# B&R Automation Studio project mappFramework
Automation Studio 4.10.4.38 SP; technology packages: mapp 5.16.1, mappCockpit 5.16.0, mappControl 5.16.0, mappFramework 1.0.0, mappMotion 5.16.2, mappView 5.16.1

## Configuration PPC2200

### Task classes (Cpu.sw)
```
Cyclic#1 (cycle 1600 us, tolerance 1600 us):
  MainCtrl <- MainControl.MainCtrl.prg [disabled]
  AxisMgr <- MachineControl.AxisTemplate.AxisMgr.prg [disabled]
  AppAxis_1 <- MachineControl.AppAxis_1.AppAxis_1.prg
  CrossCutte <- MachineControl.CrossCutter.CrossCutter.prg [disabled]
Cyclic#2 (cycle 3200 us, tolerance 3200 us):
  PIDControl <- MainControl.PIDControl.prg [disabled]
Cyclic#5 (cycle 25600 us, tolerance 25600 us):
  ProcessCon <- Infrastructure.SysServices.ProcessConfig.prg [disabled]
  AlarmMgr <- Infrastructure.AlarmX.AlarmMgr.prg
  FileMgr <- Infrastructure.File.FileMgr.prg
  ReportMgr <- Infrastructure.Report.ReportMgr.prg
  AuditMgr <- Infrastructure.Audit.AuditMgr.prg
  UserXMgr <- Infrastructure.UserX.UserXMgr.prg
  DataMgr <- Infrastructure.Data.DataMgr.prg
  RecipeMgr <- Infrastructure.Recipe.RecipeMgr.prg
  UsbMgr <- Infrastructure.Usb.UsbMgr.prg
  BackupMgr <- Infrastructure.Backup.BackupMgr.prg
Cyclic#8 (cycle 9600 us):
  IoBrowser <- Infrastructure.SysServices.IoBrowser.prg
  SysServs <- Infrastructure.SysServices.SysServs.prg
DataObjects: McAcpSys
NcDataObjects: McDriveLog
Binaries: TCData, OpcUaSrv, McAcpSim, mCoWebSc, McProfGen, udbdef, TCLang, McAcpDrv, mvLoader, arsvcreg, arflatprv, FWRules, arcoal, sysconf, CutterAlm, asfw, UserXlogin, MachineGrp, Role, User, Settings, ashwd, ashwac, CutVirt, iomap, arconfig, CutAxis, CutCamAut, myUnits, CutterGrp, TC, BackupFile, Config, RecipeXML, AlarmXHist, RecipeCSV, VAppAxis1, Axis1Alm, Axis1Grp, AppAxis1, RecipeFile, DataFile, ReportFile, AuditFile, AuditCfg, FileCfg, BackupCfg, AlarmXCfg, ReportCfg, UserXCfg, DataCfg, Report, Audit, Data, Backup, UserX, AlarmX, Recipe, McMechSys, ConvVirt, ConvAxis, ConvGrp, ConvAlm, Cutter, AlmHistory, Rcp, Alarm, UsX
Libraries: operator, runtime, astime, AsIecCon, brsystem, sys_lib, AsArSdm, FileIO, standard, AsBrStr, asstring, AsBrWStr, ArUser, AsMem, AsARCfg, MTTypes, AsZip, DataObj, AsUPS, AsIO, AsIOMMan, Gat, IoMapMan, ArCfgMan, MTBasics, AsUSB, CoTrace, MpFile, MpData, MpBase, MpAxis, MpWebXs, MpAudit, MpRecipe, MpUserX, MpReport, MpAlarmX, MpCom, MpBackup, McAxis, McBase, McAcpAx, McPureVAx, McAcpPar, MpServer, MpRegMark, dvframe, AsIODiag, aseth, arssl, asepl, powerlnk, ashw, arproject, arcert, LoggingLib, snprintf, asarlog, asarprof
```

### Hardware
```
5AP1130.185C-000 : 5AP1130.185C-000 v2.0.0.0
5PPC2200_AL14_000 : 5PPC2200.AL14-000 v2.0.1.0  [SY -> 5AP1130.185C-000.SY1]
  Connector IF3:
    AssignedOperatingSystem = ARemb
    ActivateDevice = 1
    ActivateSnmp = 1
  Connector IF4:
    AssignedOperatingSystem = GPOS
  Connector IF7:
    OperatingSystem = ARemb
    ActivateDevice = 1
  Connector IF5:
    AssignedOperatingSystem = ARemb
  Connector IF6:
    AssignedOperatingSystem = GPOS
  ConfigurationID = mappFW_PPC2200
  UserPartitionSize = 128
  Simulation = 1
  SystemTick = 1600
  TaskClassIdleTime = 1600
  Cyclic1Duration = 1600
  Cyclic1Tolerance = 1600
  Cyclic2Duration = 3200
  Cyclic2Tolerance = 3200
  Cyclic3Duration = 6400
  Cyclic3Tolerance = 6400
  Cyclic4Duration = 12800
  Cyclic4Tolerance = 12800
  Cyclic5Duration = 25600
  Cyclic5Tolerance = 25600
  Cyclic6Duration = 51200
  Cyclic6Tolerance = 51200
  Cyclic7Duration = 102400
  Cyclic7Tolerance = 102400
  Cyclic8Duration = 9600
  FileDevice1
  FileDeviceName1 = UserPartition
  FileDevicePath1 = F:\
  FileDevice2
  FileDeviceName2 = mappRecipeFiles
  FileDevicePath2 = F:\Recipe
  FileDevice3
  FileDeviceName3 = mappAuditFiles
  FileDevicePath3 = F:\Audit
  FileDevice4
  FileDeviceName4 = mappReportFiles
  FileDevicePath4 = F:\Report
  FileDevice5
  FileDeviceName5 = mappDataFiles
  FileDevicePath5 = F:\Data
  FileDevice6
  FileDeviceName6 = mappBackupFiles
  FileDevicePath6 = F:\Backup
  FileDevice7
  FileDeviceName7 = mappAlarmXFiles
  FileDevicePath7 = F:\AlarmX
  FileDevice8
  FileDeviceName8 = mappUserXFiles
  FileDevicePath8 = F:\UserX
  TimeZone = 65
  ActivateDaylightSavingTime = 1
  FtpUser1
  FtpUsername1 = user
  FtpUserPassword1 = sHpIbnZIAriJzdWitYyNPul7Ws1MiS3ggYkn5Z1jgCk=
  FtpUserSalt1 = 13A/KPuX
  FTPAccessRight1 = 0
  FTPdevice1 = ALL
  ActivateOpcUa = 1
  OpcUaInformationModels_PV_Version = 1
  ActivateHypervisor = 1
```

### VAppAxis1.purevaxcfg - 5PPC2200_AL14_000/mappMotion/AppAxis_1/VAppAxis1.purevaxcfg
```
Element gMpLinkPureVAxCfgAppAxis_1 (Type=purevaxcfg)
  TypeID = PureVAxConfig
  PureVAxis:
    AxisReference = gMpLinkAppAxis_1
    Homing:
      Mode = Direct
        Position = 0.0
        ReferencePulse = NotUsed
      RestorePositionVariable
    JerkFilter = NotUsed
```

### CutVirt.purevaxcfg - 5PPC2200_AL14_000/mappMotion/CrossCutter/CutVirt.purevaxcfg
```
Element PureVAxCfg_CrossCutter (Type=purevaxcfg)
  TypeID = PureVAxConfig
  PureVAxis:
    AxisReference = gAxisCrossCutter
    Homing:
      Mode = Direct
        Position = 0.0
        ReferencePulse = NotUsed
      RestorePositionVariable
    JerkFilter = NotUsed
```

### Axis1Grp.mpcomgroup - 5PPC2200_AL14_000/mappServices/AppAxis_1/Axis1Grp.mpcomgroup
```
Element gMpLinkGroupAppAxis_1 (Type=mpcomgroup)
  Linking:
    Subnodes:
      0 = gMpLinkAppAxis_1
      1 = gMpLinkAlarmXCoreAppAxis_1
  Alarms = MpAlarmX
```

### BackupFile.mpfilemanagerui - 5PPC2200_AL14_000/mappServices/Backup/BackupFile.mpfilemanagerui
```
Element gMpLinkFileManagerUIBackup (Type=mpfilemanagerui)
  Alarms = MpAlarmX
    mapp.AlarmX.Core.Configuration:
      [0]:
        Message = {$File/Alarms/DeviceNotFound}
      [1]:
        Message = {$File/Alarms/AlreadyExisting}
      [2]:
        Message = {$File/Alarms/FileSystemError}
```

### CutterGrp.mpcomgroup - 5PPC2200_AL14_000/mappServices/CrossCutter/CutterGrp.mpcomgroup
```
Element gGroupCutter (Type=mpcomgroup)
  Linking:
    Subnodes:
      0 = gAxisCrossCutter
      1 = gAlarmXCore_Cutter
  Alarms = MpAlarmX
```

### FileCfg.mpfilemanagerui - 5PPC2200_AL14_000/mappServices/File/FileCfg.mpfilemanagerui
```
Element gMpLinkFileManagerUIFile (Type=mpfilemanagerui)
  Alarms = MpAlarmX
    mapp.AlarmX.Core.Configuration:
      [0]:
        Message = {$File/Alarms/DeviceNotFound}
      [1]:
        Message = {$File/Alarms/AlreadyExisting}
      [2]:
        Message = {$File/Alarms/FileSystemError}
```

### RecipeXML.mprecipexml - 5PPC2200_AL14_000/mappServices/Recipe/RecipeXML.mprecipexml
```
Element gMpLinkRecipeXml (Type=mprecipexml)
  mapp.Recipe.Xml:
    Auditing = MpAudit
  Alarms = MpAlarmX
    mapp.AlarmX.Core.Configuration:
      [0]:
        Message = {$Recipe/Alarms/SaveFailed}
      [1]:
        Message = {$Recipe/Alarms/SaveFailedPartial}
        Disable = TRUE
      [2]:
        Message = {$Recipe/Alarms/LoadFailed}
      [3]:
        Message = {$Recipe/Alarms/LoadFailedPartial}
        Disable = TRUE
```

### ReportCfg.mpreportcore - 5PPC2200_AL14_000/mappServices/Report/ReportCfg.mpreportcore
```
Element gMpLinkReport (Type=mpreportcore)
  MpReport:
    Settings:
      ResourceDeviceName = mappReport
      LanguageDependent:
        [0]:
          Language = en
          Font = 1
        [1]:
          Language = zh-CN
    PageLayouts:
      [0]:
        Name = Default
    Styles:
      Text:
        [0]:
          Name = Default
          Size = 12
        [1]:
          Name = Header
          Style = 1
          Size = 20
          Color = FF9900
        [2]:
          Name = Subheader
          Size = 16
          Color = FF9900
      Table:
        [0]:
          Name = Default
          Padding = 10
      Line:
        [0]:
          Name = Default
          Color = FF9900
      Chart:
        PieChart:
          [0]:
            Name = Default
            BorderWidth = 0
        LineChart:
          [0]:
            Name = Default
        BarChart:
          [0]:
            Name = Default
    Tables:
      [0]:
        Name = Information
        TableStyle = Default
        TextStyle = Default
        [0]:
          [0] = TextId
            Source = RecipeName
            Width = 50
          [1] = ValueId
            Value:
              ProcessVariable = ::RecipeMgr:MpRecipe_0.Info.LastLoadedRecipe
            Width = 50
        [1]:
          [0] = TextId
            Source = Index
            Width = 50
          [1] = TextId
            Source = Length [mm]
            Width = 50
          [2] = TextId
            Source = Number
            Width = 50
        [2]:
          [0] = TextId
            Source = 1
            Width = 50
          [1] = ValueId
            Value:
              ProcessVariable = ::MainCtrl:MainCtrl.Para.ProductLength[0]
            Width = 50
          [2] = ValueId
            Value:
              ProcessVariable = ::MainCtrl:MainCtrl.Para.ProductNumber[0]
            Width = 50
        [3]:
          [0] = TextId
            Source = 2
            Width = 50
          [1] = ValueId
            Value:
              ProcessVariable = ::MainCtrl:MainCtrl.Para.ProductLength[1]
            Width = 50
          [2] = ValueId
            Value:
              ProcessVariable = ::MainCtrl:MainCtrl.Para.ProductNumber[1]
            Width = 50
        [4]:
          [0] = TextId
            Source = 3
            Width = 50
          [1] = ValueId
            Value:
              ProcessVariable = ::MainCtrl:MainCtrl.Para.ProductLength[2]
            Width = 50
          [2] = ValueId
            Value:
              ProcessVariable = ::MainCtrl:MainCtrl.Para.ProductNumber[2]
            Width = 50
        [5]:
          [0] = TextId
            Source = 4
            Width = 50
          [1] = ValueId
            Value:
              ProcessVariable = ::MainCtrl:MainCtrl.Para.ProductLength[3]
            Width = 50
          [2] = ValueId
            Value:
              ProcessVariable = ::MainCtrl:MainCtrl.Para.ProductNumber[3]
            Width = 50
        [6]:
          [0] = TextId
            Source = 5
            Width = 50
          [1] = ValueId
            Value:
              ProcessVariable = ::MainCtrl:MainCtrl.Para.ProductLength[4]
            Width = 50
          [2] = ValueId
            Value:
              ProcessVariable = ::MainCtrl:MainCtrl.Para.ProductNumber[4]
            Width = 50
    Contents:
      [0]:
        Name = ContentHeader
        [0]:
          Text = {Header}
        [1] = DateTime
        [2] = Line
          LineStyle = Default
      [1]:
        Name = ContentTable
        [0] = Table
          Table = Information
          HorizontalAlign = 1
      [2]:
        Name = Header
        [0]:
          Text = Report of the Cross Cutter Machine
          HorizontalAlign = 1
          TextStyle = Header
      [3]:
        Name = EmptyLine
        [0] = EmptyLine
      [4]:
        Name = Underline
        [0] = Line
          LineStyle = Default
      [5]:
        Name = Date
        [0] = DateTime
          TextStyle = Default
    Reports:
      [0]:
        Name = Report
        PageLayout = Default
        Header = Header
        [0]:
          [0]:
            Content = Underline
        [1]:
          [0]:
            Content = EmptyLine
        [2]:
          Heading:
            Text = Time
            TextStyle = Subheader
          [0]:
            Content = Date
        [3]:
          [0]:
            Content = EmptyLine
        [4]:
          [0]:
            Content = EmptyLine
        [5]:
          Heading:
            Text = Data
            TextStyle = Subheader
          [0]:
            Content = ContentTable
  Alarms = MpAlarmX
    mapp.AlarmX.Core.Configuration:
      [0]:
        Message = {$Report/Alarms/GenerateFailed}
```

## Configuration TS_UnitTest_Sample

CPU , AutomationRuntime D4.91, Build 6.3.0, Safety 0.0

### Hardware
```
PC_any : PC_any v1.1.1.0 (OrderNumber=PC)
  ConfigurationID = GAT_TS_UnitTest_Sample
  Cyclic1Duration = 10000
  Cyclic8Duration = 10000
  ActivateOpcUa = 1
  OpcUaInformationModels_PV_Version = 1
```

### AxisTest.vvm - PC_any/AxisTest.vvm
```iecst
VAR_CONFIG
	::prototypeT:AxisControl.Command AT %Q.::AxisContro:AxisControl.Command; (*Insert your comment here...*)
	::prototypeT:AxisControl.Parameters AT %Q.::AxisContro:AxisControl.Parameters; (*Insert your comment here...*)
	::AxisContro:AxisControl.Status AT %Q.::prototypeT:AxisControl.Status; (*Insert your comment here...*)
END_VAR
```

### Cutter.regmarkdetection - PC_any/mappControl/Cutter.regmarkdetection
```
Element gRegMarkDetection_Cutter (Type=regmarkdetection)
  RegistrationMarkDetection:
    SensorSignal:
      AxisReference = gAxisCrossCutter
      DelayCompensation:
        AdditionalDelayTime  // 0.
    Measurement = MarkToCylinder
      Product:
        Position:
          AxisReference = gAxisAppAxis_1
          Source = SetValue
        Length:
          Value = 70
    Detection = MiddleOfEdges
      SetMarkPosition = 0
      ExpectationWindow:
        Width = 25
      MarkWidthMonitoring:
        MinimumWidth = 7
        MaximumWidth = 15
      MissedMarkReaction:
        MarkPosition = LastValue
        AutomaticSearch = Used
          AdditionalExpectationWindowShift = 25
    OutputSignals:
      ActualMarkPosition = ::CrossCutte:RegistrationControl.ActualMarkPosition
      MarkPositionError = ::CrossCutte:RegistrationControl.MarkPositionError
      ActualProductLength = ::CrossCutte:RegistrationControl.ActualProductLength
      ActualIntervalLength = ::CrossCutte:RegistrationControl.ActualIntervalLength
  Alarms = MpAlarmX
```

### TestAlm.mpalarmxcore - PC_any/mappServices/AxisTest/TestAlm.mpalarmxcore
```
Element gAlarmXCore_Test (Type=mpalarmxcore)
  mapp.AlarmX.Core:
    BySeverity:
      [0]:
        Severity = 1..9
        [0] = Reaction
          Name = Info
        [1] = Escalate
      [1]:
        Severity = 10..19
        [0] = Reaction
          Name = Error
        [1] = Escalate
      [2]:
        Severity = 20..29
        [0] = Reaction
          Name = Error
        [1] = Escalate
        [2] = EscalateReaction
          Reaction = Error
      [3]:
        Severity = 30..39
        [0] = Reaction
          Name = Safety
        [1] = Escalate
        [2] = Remain
    Default:
      [0] = Reaction
        Name = Duplicate
      [1] = Escalate
      [2] = Remain
  mapp.AlarmX.Core.Configuration:
    [0]:
      Name = ReferenceRequired
      Message = {$IAT/Axis/Info/Name} : {$IAT/Axis/Alarms/ReferenceRequired}
      Severity = 10
      Behavior = DiscreteValueMonitoring
        Monitoring:
          MonitoredPV = ::AxisContro:AxisControl.Status.ReferenceRequired
          TriggerValues:
            [0] = 1
```

## Logical view

Binary libraries used (declarations not repeated): UtMgr 2.01.0, UtWs 2.01.0, ArCfgMan 1.01.1, ArUser, AsARCfg, AsBrStr, AsBrWStr, AsIecCon, AsIO, AsIODiag, AsIOMMan, asstring, AsUPS, AsUSB, AsZip, brsystem, CoTrace, DataObj, dvframe, FileIO, IoMapMan 1.01.1, McAcpAx 5.16.2, McAcpPar 5.16.2, McAxis, McPureVAx 5.16.2, MpAlarmX 5.16.1, MpAudit 5.16.1, MpAxis, MpBackup 5.16.1, MpBase 5.16.0, MpCom 5.16.1, MpData 5.16.1, MpFile 5.16.1, MpRecipe, MpRegMark 5.16.0, MpReport 5.16.1, MpServer 5.16.0, MpUserX 5.16.1, MpWebXs 5.16.1, MTBasics 5.16.0, MTTypes 1.03.4, operator, runtime, standard, sys_lib

### mappFrameworkGlobal.var
```iecst
VAR CONSTANT
	PARAMETERS_CATEGORY : STRING[10] := 'Parameters'; (*Recipe category for runtime parameters*)
	MACHINE_CONFIGURATION_CATEGORY : STRING[30] := 'Machine Configuration'; (*Recipe category for machine configuration settings*)
	MAX_IDX_USB_DEV_LIST : USINT := 1; (*Maximum number of USB storage devices. Value 1 = 2 USB devices (index 0 and 1)*)
END_VAR
VAR
	gUSBAvailable : ARRAY[0..MAX_IDX_USB_DEV_LIST] OF BOOL; (*Boolean array for whether the USB device is plugged in*)
END_VAR
```

- Project.language (not shown)

### Program Logical/Infrastructure/AlarmX/AlarmMgr (IEC) - Alarm manager

#### ExecuteQuery.st
```iecst
ACTION ExecuteQuery:

	// Initialize mapp function block
	QueryActiveAlarms_0.MpLink := ADR(gMpLinkAlarmXCore);
	QueryActiveAlarms_0.Enable := TRUE;
	QueryActiveAlarms_0.Name := ADR('ActiveAlarms');
	QueryActiveAlarms_0.Language := ADR('en');
	QueryActiveAlarms_0();

	CASE (AlarmQuery.State) OF
		ACTIVE_ALARM_WAIT:
			// Wait until the RunQuery command is triggered from the HMI.
			// If you prefer that the query runs anytime new data is available, then uncomment line 15 and comment out line 16 and delete
			// the "Run query" button from the HMI.
			//IF (AlarmQuery.LastUpdateCount <> AlarmQuery.UpdateCount) THEN
			IF (HmiAlarmX.Commands.RunQuery = TRUE) THEN
				brsmemset(ADR(AlarmQuery.Alarms[0]), 0, SIZEOF(AlarmQuery.Alarms));
				AlarmQuery.LastUpdateCount := AlarmQuery.UpdateCount;
				QueryActiveAlarms_0.Execute := TRUE;
				HmiAlarmX.Commands.RunQuery := FALSE;
				AlarmQuery.State := ACTIVE_ALARM_QUERY;
			END_IF

		ACTIVE_ALARM_QUERY:
			// If the number of query results is less than MAX_QUERY_RESULTS, return to the wait state
			IF ((QueryActiveAlarms_0.CommandDone = TRUE) AND (QueryActiveAlarms_0.Info.HasMoreRows = FALSE)) THEN
				QueryActiveAlarms_0.Execute := FALSE;
				QueryActiveAlarms_0.Next := FALSE;
				AlarmQuery.State := ACTIVE_ALARM_WAIT;
				// If the number of query results is more than MAX_QUERY_RESULTS, then query the next set of results
			ELSIF ((QueryActiveAlarms_0.CommandDone = TRUE) AND (QueryActiveAlarms_0.Info.HasMoreRows = TRUE)) THEN
				QueryActiveAlarms_0.Next := FALSE;
				AlarmQuery.State := ACTIVE_ALARM_NEXT;
			END_IF

		ACTIVE_ALARM_NEXT:
			IF (AlarmQuery.Next = TRUE) THEN
				// By default, AlarmQuery.Alarms has 20 elements, so it can hold 20 query results at a time (MAX_QUERY_RESULTS = 19).
				// If AlarmQuery.Next is true, this means the query result is more than 20 alarms.
				// If you want to save the data for the first 20 alarms, add code here to copy AlarmQuery.Alarms to another location.
				// Otherwise, the older alarms in the query will get overwritten with the newest entries here.
				brsmemset(ADR(AlarmQuery.Alarms[0]), 0, SIZEOF(AlarmQuery.Alarms));
				AlarmQuery.Next := FALSE;
				QueryActiveAlarms_0.Next := TRUE;
				AlarmQuery.State := ACTIVE_ALARM_QUERY;
			END_IF
	END_CASE

	// Convert the query results into arrays that can easily be bound to the Table widget in mapp View
	FOR i := 0 TO MAX_QUERY_RESULTS DO
		HmiAlarmX.Status.Query.Active[i] := AlarmQuery.Alarms[i].Active;
		HmiAlarmX.Status.Query.Acknowledged[i] := AlarmQuery.Alarms[i].Acknowledged;
		HmiAlarmX.Status.Query.Scope[i] := AlarmQuery.Alarms[i].Scope;
		HmiAlarmX.Status.Query.Name[i] := AlarmQuery.Alarms[i].Name;
		HmiAlarmX.Status.Query.Message[i] := AlarmQuery.Alarms[i].Message;
		HmiAlarmX.Status.Query.AdditionalInfo[i] := AlarmQuery.Alarms[i].AdditionalInfo;
		HmiAlarmX.Status.Query.TimeStamp[i] := AlarmQuery.Alarms[i].TimeStamp;
		HmiAlarmX.Status.Query.Severity[i] := AlarmQuery.Alarms[i].Severity;
	END_FOR

END_ACTION
```

- Program Logical/Infrastructure/Audit/AuditMgr (IEC) (no source held here)

### Program Logical/Infrastructure/Backup/BackupMgr (IEC) - Backup manager

#### BackupMgr.typ
```iecst
(*Structure types*)

TYPE
	BackupHmiInterfaceType : 	STRUCT  (*HMI interface structure*)
		Commands : BackupHmiCommandsType; (*Structure to hold the commands from the HMI*)
		Parameters : BackupHmiParametersType; (*Structure to hold the parameters for the HMI*)
		Status : BackupHmiStatusType; (*Structure to hold the status information from the HMI*)
	END_STRUCT;
	BackupHmiCommandsType : 	STRUCT  (*Structure to hold the commands from the HMI*)
		Create : BOOL; (*Create a backup*)
		Restore : BOOL; (*Restore a backup*)
		Delete : BOOL; (*Delete a backup*)
		SaveConfig : BOOL; (*Save automatic backup configuration settings*)
		Reset : BOOL; (*Error reset*)
	END_STRUCT;
	BackupHmiParametersType : 	STRUCT  (*Structure to hold the parameters for the HMI*)
		Name : STRING[80] := 'myBackup'; (*Name of the backup*)
		AutomaticBackup : AutomaticBackupType; (*Automatic backup settings*)
	END_STRUCT;
	BackupHmiStatusType : 	STRUCT  (*Structure to hold the status information from the HMI*)
		Busy : BOOL; (*Backup is busy executing an action*)
		Error : BOOL; (*Error flag*)
		CreateAllowed : BOOL; (*Bit to indicate it is allowable to create a backup right now*)
		RestoreAllowed : BOOL; (*Bit to indicate it is allowable to restore a backup right now*)
		FileNames : ARRAY[0..49]OF STRING[80]; (*Existing backup file names*)
		TimeStamps : ARRAY[0..49]OF DATE_AND_TIME; (*Time stamps for existing backups*)
		Size : {REDUND_UNREPLICABLE} ARRAY[0..49]OF UDINT; (*Sizes of existing backup files*)
		Info : MpBackupProjectInfoRequestType; (*Project information (name, configuration ID, configuration version)*)
		DeviceDataProvider : ARRAY[0..MAX_IDX_FILE_DEV]OF STRING[100]; (*Data provider for file device dropdown on automatic backup configuration pop-up*)
		TableConfig : ARRAY[0..1]OF STRING[120]; (*Table configuration for the list of available backups*)
		SimulationActive : BOOL; (*Flag for if simulation is active*)
		SelectedIndex : USINT; (*Index of the selected backup file*)
		LastSelectedIndex : USINT; (*Index of the last selected backup file*)
		LastSelectedDeviceIndex : UINT; (*Index of the last selected file device. Compared with MpFileManagerUIConnect.DeviceList.SelectedIndex*)
	END_STRUCT;
	AutomaticBackupType : 	STRUCT  (*Automatic backup settings*)
		Enable : BOOL; (*Enable automatic backup feature*)
		Prefix : STRING[50]; (*Name prefix for each automatic backup file*)
		Device : STRING[255]; (*File device to store the automatic backup*)
		Mode : AutomaticBackupModeType; (*Automatic backup time interval*)
		OverwriteOldest : MpBackupOverwriteOldestType; (*Defines whether older backups should be deleted or not*)
	END_STRUCT;
	AutomaticBackupModeType : 	STRUCT  (*Automatic backup time interval*)
		Interval : AutomaticBackupIntervalEnum; (*Day interval (daily, or a specfiic day of the week)*)
		Hour : USINT; (*Time (hour)*)
		Minute : USINT; (*Time (minutes)*)
	END_STRUCT;
END_TYPE

(*Enumerations*)

TYPE
	AutomaticBackupIntervalEnum :
		( (*Selection for how often to automatically create a backup*)
		BACKUP_EVERYDAY, (*Every day*)
		BACKUP_MONDAY, (*Every Monday*)
		BACKUP_TUESDAY, (*Every Tuesday*)
		BACKUP_WEDNESDAY, (*Every Wednesday*)
		BACKUP_THURSDAY, (*Every Thursday*)
		BACKUP_FRIDAY, (*Every Friday*)
		BACKUP_SATURDAY, (*Every Saturday*)
		BACKUP_SUNDAY (*Every Sunday*)
		);
	BackupStateEnum :
		( (*States for backup state machine*)
		BACKUP_IDLE, (*Wait state*)
		BACKUP_CREATING, (*Creating a backup*)
		BACKUP_RESTORING, (*Restoring a backup*)
		BACKUP_DELETING, (*Deleting a backup*)
		BACKUP_ERROR (*Error state*)
		);
END_TYPE
```

#### ChangeConfiguration.st
```iecst
ACTION ChangeConfiguration:

    MpBackupCoreConfig_0.MpLink := ADR(gMpLinkBackupCore);
    MpBackupCoreConfig_0.Configuration := ADR(MpBackupConfiguration);
    IF (MpBackupCoreConfig_0.Error = TRUE) THEN
        // Loading currently always throws an error about failed to write Auditing.Type
        IF (MpBackupCoreConfig_0.StatusID = mpBACKUP_ERR_CONFIG_LOAD) THEN
            LoadBackupConfiguration;
        END_IF

        MpBackupCoreConfig_0.Load := FALSE;
        MpBackupCoreConfig_0.Save := FALSE;
        MpBackupCoreConfig_0.ErrorReset := TRUE;
    END_IF
    MpBackupCoreConfig_0();
    MpBackupCoreConfig_0.ErrorReset := FALSE;
    IF (MpBackupCoreConfig_0.CommandDone = TRUE) THEN
        IF (MpBackupCoreConfig_0.Load = TRUE) THEN
            LoadBackupConfiguration;
        END_IF
        MpBackupCoreConfig_0.Load := FALSE;
        MpBackupCoreConfig_0.Save := FALSE;
    END_IF

END_ACTION
```

### Program Logical/Infrastructure/Data/DataMgr

#### DataMgr.st
```iecst
//*********************************************************************************
//* Copyright: B&R Industrial Automation GmbH
//* Author:    B&R Industrial Automation GmbH
//* Created:   30. Sep 2020/08:00
//* Description: Tasks FOR Data Management control. The Data Management handling is done in this task.
//*********************************************************************************

PROGRAM _INIT

	// Create folder for this component on the user file device
	DirCreate_0(enable := TRUE, pDevice := ADR('UserPartition'), pName := ADR(LOCAL_FOLDER));

	// Check if folder already exist and if so disabled the function block call
	IF DirCreate_0.status = fiERR_DIR_ALREADY_EXIST THEN
		DirCreate_0(enable := FALSE);
	END_IF

	// Init mapp function blocks
	MpFileManagerUI_0.Enable := TRUE;
	MpFileManagerUI_0.MpLink := ADR(gMpLinkFileManagerUIData);
	MpFileManagerUI_0.UIConnect := ADR(MpFileManagerUIConnect);

	MpDataRecorder_0.MpLink := ADR(gMpLinkDataRecorder);
	MpDataRecorder_0.Enable := TRUE ;
	MpDataRecorder_0.DeviceName := ADR('mappDataFiles');
	MpDataRecorder_0.RecordMode := mpDATA_RECORD_MODE_TIME;
	MpDataRecorder_0.SamplingTime := t#5s;

	// Register PVs for data recording
	MpDataRegPar_x[0].MpLink := ADR(gMpLinkDataRecorder);
	MpDataRegPar_x[0].Enable := TRUE;
	MpDataRegPar_x[0].PVName := ADR('PIDControl:rActValue');
	MpDataRegPar_x[0].Description := ADR('Control Value');

	MpDataRegPar_x[1].MpLink := ADR(gMpLinkDataRecorder);
	MpDataRegPar_x[1].Enable := TRUE;
	MpDataRegPar_x[1].PVName := ADR('MainCtrl:MpAxisBasic_x[0].Velocity');
	MpDataRegPar_x[1].Description := ADR('Feeder Velocity');

	// Filter files for pdf type
	MpFileManagerUIConnect.File.Filter := '*.pdf';
END_PROGRAM

PROGRAM _CYCLIC
	//***************************************************
	FOR i := 0 TO 49 DO
		// Save Filenames to a seperate array for display in Table
		DisplayFileName[i] := MpFileManagerUIConnect.File.List.Items[i].Name;
		// Mark file selection
		MpFileManagerUIConnect.File.List.Items[i].IsSelected := (DisplayFileNameIndex = INT_TO_USINT(i));
    END_FOR
    // String for pdfViewer to display right report
	StrSelectedFile := CONCAT(STR_FILE_DEVICE, MpFileManagerUIConnect.File.List.Items[DisplayFileNameIndex].Name);

	// Configure visible file list
	brsstrcpy(ADR(TableConfig), ADR('{ "specRows": [{"from":'));
	brsitoa(MpFileManagerUIConnect.File.PathInfo.FileCount, ADR(TableConfig) + brsstrlen(ADR(TableConfig)));
	brsstrcat(ADR(TableConfig),  ADR(',"to":49, "visible":false}]}'));

	// Call function blocks
	MpDataRecorder_0();
	FOR i := 0 TO MAX_IDX_DATA_REG DO
		MpDataRegPar_x[i]();
	END_FOR
	MpFileManagerUI_0();

	// Reset ErrorReset command
	IF NOT MpDataRecorder_0.Error THEN
		MpDataRecorder_0.ErrorReset := FALSE;
	END_IF
	FOR i := 0 TO MAX_IDX_DATA_REG DO
		IF NOT MpDataRegPar_x[i].Error THEN
			MpDataRegPar_x[i].ErrorReset := FALSE;
		END_IF
	END_FOR
END_PROGRAM

PROGRAM _EXIT
	// Call mapp function blocks with enable = false
	MpFileManagerUI_0.Enable := FALSE;
	MpFileManagerUI_0();
	MpDataRecorder_0.Enable := FALSE;
	MpDataRecorder_0();
	FOR i := 0 TO MAX_IDX_DATA_REG DO
		MpDataRegPar_x[i].Enable := FALSE;
		MpDataRegPar_x[i]();
	END_FOR
END_PROGRAM
```

### Program Logical/Infrastructure/File/FileMgr (IEC)

#### FileMgr.typ - Local data types
```iecst
(*Structure types*)

TYPE
	FileHmiInterfaceType : 	STRUCT  (*Structure to hold commands, parameters and status from the HMI*)
		Commands : FileHmiCommandsType; (*Structure to hold the commands from the HMI*)
		Parameters : FileHmiParametersType; (*Structure to hold parameters for the mapp View HMI*)
		Status : FileHmiStatusType; (*Structure to hold status information from the mapp View HMI*)
	END_STRUCT;
	FileHmiCommandsType : 	STRUCT  (*Structure to hold the commands from the HMI*)
		Delete : BOOL; (*Delete file*)
		FolderUp : BOOL; (*Move back/up a folder*)
		EnterFolder : BOOL; (*Move forward/down a folder*)
		MultiSelect : BOOL; (*Enables the ability to select multiple files*)
		CheckFolder : BOOL; (*Run the FIFO check to determine if old files should be deleted*)
	END_STRUCT;
	FileHmiParametersType : 	STRUCT  (*Structure to hold parameters for the mapp View HMI*)
		OldSortOrder : MpFileManagerUISortOrderEnum; (*Previous sord order*)
		Fifo : FileHmiParaFifoType; (*Parameters for the FIFO feature (first-in-first-out)*)
	END_STRUCT;
	FileHmiStatusType : 	STRUCT  (*Structure to hold status information from the mapp View HMI*)
		FileNames : ARRAY[0..49]OF STRING[80]; (*List of file names*)
		TimeStamps : ARRAY[0..49]OF DATE_AND_TIME; (*List of time stamps for file names*)
		Type : ARRAY[0..49]OF DINT; (*List of file types*)
		Size : ARRAY[0..49]OF UDINT; (*List of file sizes*)
		DeviceDataProvider : ARRAY[0..MAX_IDX_FILE_DEV]OF STRING[100]; (*Data provider for the file device selector*)
		DeviceName : STRING[50]; (*File device name*)
		FileName : STRING[255]; (*Fille name*)
		TableConfig : ARRAY[0..1]OF STRING[120]; (*Table configuration for the file explorer (table widget) on the mapp View HMI*)
		IsFolder : BOOL; (*Flag for whether the item is a folder (versus a file)*)
		BackButton : BOOL; (*Flag for whether the back button should be shown*)
		DeleteStep : FileDeleteStepEnum; (*Enumeration for automatic file deletion steps*)
		AutoDeleteSelected : USINT; (*Number of selected items*)
		FolderSize : REAL; (*Size of currently selected folder*)
		SelectedIndex : USINT; (*Selected index in the file list*)
		CurrentPage : STRING[80]; (*Current page*)
	END_STRUCT;
	FileHmiParaFifoType : 	STRUCT  (*Parameters for the FIFO feature (first-in-first-out)*)
		Enable : BOOL; (*FIFO enable*)
		DeviceName : STRING[50]; (*File device that the FIFO is active on*)
		FifoType : FileFifoTypeEnum; (*Defines the delete behavior of the FIFO*)
		ScanInterval : DINT := 60; (*[minutes]*)
		MaxFileAge : UINT := 365; (*[days] Files older than 1 year will be deleted*)
		MaxFolderSize : REAL := 1000; (*[kB] - Max size of files inside the active folder*)
		MaxNumberOfFiles : UINT := 20; (*Max number of files inside active folder*)
	END_STRUCT;
	FilePathCheckType : 	STRUCT  (*Setup for checking available folders / file devices for FIleManager*)
		Folder : ARRAY[0..9]OF STRING[20]; (*Folder name in user partition*)
		DeviceList : MpFileManagerUIDeviceListType; (*Device name*)
	END_STRUCT;
END_TYPE

(*Enumerations*)

TYPE
	FileDeleteStepEnum :
		( (*Enumeration for file deletion steps*)
		FILE_DELETE_WAIT := 0, (*Wait state*)
		FILE_SCAN_FOLDER_WAIT, (*Wait for check for old files command*)
		FILE_SELECT_DEVICE, (*Switch file device to the configured one *)
		FILE_SORT_BY_DATE, (*Sort by date so the oldest files are at the end*)
		FILE_SORT_BY_DATE_WAIT, (*Wait step switching sorting mode*)
		FILE_CHECK_FOR_FILTER, (*Check which delete filter is active*)
		FILE_SELECT_OLDEST_FILES_0, (*Scan and select all file over the filter setting*)
		FILE_CALC_FOLDER_SIZE, (*Calculate the overall file size in the open folder*)
		FILE_SELECT_OLDEST_FILES_1, (*Scan and select all file over the filter setting*)
		FILE_DELETE_FILES, (*Set command to delete the selected oldest files*)
		FILE_CONFIRM_DELETE, (*Confirm the file delete*)
		FILE_RESET_SORT_BY, (*Restore old sort order*)
		FILE_RESET_SORT_BY_WAIT (*Waiting for restore previous sort order*)
		);
	FileFifoTypeEnum :
		( (*Defines the delete behavior of the FIFO*)
		FILE_FIFO_NUM_OF_FILES := 0, (*Delete according to total number of files*)
		FILE_FIFO_SIZE_OF_FOLDER (*Delete according to maximum folder size*)
		);
	FileTypeEnum :
		( (*Defines the type of file in order to update the displayed icon*)
		FOLDER := 0, (*Folder*)
		FILE := 1, (*File*)
		FILE_SELECTED := 2 (*The selected file*)
		);
END_TYPE
```

#### HMIActions.st - Supporting code for the HMI interface
```iecst
ACTION FormatDeviceDataProvider:

	// Select CF device if USB device is not available
    FOR i := 0 TO MAX_IDX_USB_DEV_LIST DO
        IF gUSBAvailable[i] THEN

			HmiFile.Status.DeviceDataProvider[i + USBOffset] := '{"value":"USB';
            brsitoa(i + 1, ADR(HmiFile.Status.DeviceDataProvider[i + USBOffset]) + brsstrlen(ADR(HmiFile.Status.DeviceDataProvider[i + USBOffset])));

			brsstrcat(ADR(HmiFile.Status.DeviceDataProvider[i + USBOffset]), ADR('","text":"USB'));
            brsitoa(i + 1, ADR(HmiFile.Status.DeviceDataProvider[i + USBOffset]) + brsstrlen(ADR(HmiFile.Status.DeviceDataProvider[i + USBOffset])));
            brsstrcat(ADR(HmiFile.Status.DeviceDataProvider[i + USBOffset]), ADR('"}'));

			PathCheck.DeviceList.DeviceNames[i + USBOffset] := 'USB';
			brsitoa(i + 1, ADR(PathCheck.DeviceList.DeviceNames[i + USBOffset]) + brsstrlen(ADR(PathCheck.DeviceList.DeviceNames[i + USBOffset])));
        ELSE
			brsmemset(ADR(HmiFile.Status.DeviceDataProvider[i + USBOffset]), 0, SIZEOF(HmiFile.Status.DeviceDataProvider[i + USBOffset]));
            brsmemset(ADR(PathCheck.DeviceList.DeviceNames[i + USBOffset]), 0, SIZEOF(PathCheck.DeviceList.DeviceNames[i + USBOffset]));
        END_IF
    END_FOR

	//Check initilized folder for existance and remove any from the device list that don't exist
	IF DirInfo_0.status = ERR_OK  THEN
		IF PathCheck.DeviceList.DeviceNames[DeviceListCount] = '' THEN
			//Delete entries past the actual number of devices found
			FOR i:=Index TO 9 DO
				MpFileManagerUIConnect.DeviceList.DeviceNames[i] := '';
			END_FOR
			Index := -1;
			DeviceListCount := -1;
		END_IF
		// copy device name from source list into the actual device list
		MpFileManagerUIConnect.DeviceList.DeviceNames[Index] := PathCheck.DeviceList.DeviceNames[DeviceListCount];
		Index := Index + 1;

		DeviceListCount := DeviceListCount + 1;
		IF DeviceListCount > 9 THEN
			DeviceListCount := 0;
		END_IF
		IF Index > 9 THEN
			Index := 0;
		END_IF
	ELSIF DirInfo_0.status = fiERR_DIR_NOT_EXIST  THEN
		DeviceListCount := DeviceListCount + 1;
		IF DeviceListCount > 9 THEN
			DeviceListCount := 0;
		END_IF
	END_IF

	DirInfo_0(enable:= TRUE, pDevice := ADR('UserPartition'), pPath := ADR(PathCheck.Folder[DeviceListCount]));

	// Configure visible device list
	HmiFile.Status.TableConfig[0] := '{ "specRows": [{"from":';
	FOR i := 0 TO 9 DO
		IF MpFileManagerUIConnect.DeviceList.DeviceNames[i] <> '' THEN
			DeviceCount := i + 1;
		END_IF
	END_FOR
	brsitoa((DeviceCount), ADR(HmiFile.Status.TableConfig[0]) + brsstrlen(ADR(HmiFile.Status.TableConfig[0])));
    brsstrcat(ADR(HmiFile.Status.TableConfig[0]),  ADR(',"to":9, "visible":false}]}'));

    // Configure visible file list
	HmiFile.Status.TableConfig[1] := '{ "specRows": [{"from":';
    brsitoa((MpFileManagerUIConnect.File.PathInfo.FileCount + MpFileManagerUIConnect.File.PathInfo.FolderCount), ADR(HmiFile.Status.TableConfig[1]) + brsstrlen(ADR(HmiFile.Status.TableConfig[1])));
    brsstrcat(ADR(HmiFile.Status.TableConfig[1]),  ADR(',"to":49, "visible":false}]}'));

END_ACTION

ACTION FileManager:

    MpFileManagerUI_0.MpLink := ADR(gMpLinkFileManagerUIFile);
    MpFileManagerUI_0.UIConnect := ADR(MpFileManagerUIConnect);
	MpFileManagerUI_0();

    FOR i := 0 TO ((SIZEOF(HmiFile.Status.FileNames)/SIZEOF(HmiFile.Status.FileNames[0])) - 1) DO
        HmiFile.Status.FileNames[i] := MpFileManagerUIConnect.File.List.Items[i].Name;
        HmiFile.Status.TimeStamps[i] := MpFileManagerUIConnect.File.List.Items[i].LastModified;
        HmiFile.Status.Size[i] := REAL_TO_UDINT(UDINT_TO_REAL(MpFileManagerUIConnect.File.List.Items[i].Size) * 0.001);

		// Set image array based on item type
		IF MpFileManagerUIConnect.File.List.Items[i].IsFolder THEN
			HmiFile.Status.Type[i] := FOLDER;
		ELSIF NOT MpFileManagerUIConnect.File.List.Items[i].IsFolder AND MpFileManagerUIConnect.File.List.Items[i].IsSelected THEN
			HmiFile.Status.Type[i] := FILE_SELECTED;
		ELSE
			HmiFile.Status.Type[i] := FILE;
		END_IF

		// Set file selected when the table is clicked Single and MultiSelect
		IF HmiFile.Status.DeleteStep = FILE_DELETE_WAIT THEN
			IF (MpFileManagerUIConnect.File.MultiSelect = FALSE) THEN
				IF (i = HmiFile.Status.SelectedIndex) THEN
					MpFileManagerUIConnect.File.List.Items[i].IsSelected := TRUE;
				ELSE
					MpFileManagerUIConnect.File.List.Items[i].IsSelected := FALSE;
				END_IF
			ELSIF (MpFileManagerUIConnect.File.MultiSelect = TRUE) AND HmiFile.Commands.MultiSelect THEN
				IF (i = HmiFile.Status.SelectedIndex) AND NOT MpFileManagerUIConnect.File.List.Items[i].IsSelected THEN
					MpFileManagerUIConnect.File.List.Items[i].IsSelected := TRUE;
					HmiFile.Commands.MultiSelect := FALSE;
				ELSIF (i = HmiFile.Status.SelectedIndex) AND MpFileManagerUIConnect.File.List.Items[i].IsSelected THEN
					MpFileManagerUIConnect.File.List.Items[i].IsSelected := FALSE;
					HmiFile.Commands.MultiSelect := FALSE;
				END_IF
			END_IF
		END_IF
    END_FOR

	// Read currently selected device name for HMI
	HmiFile.Status.DeviceName := MpFileManagerUIConnect.DeviceList.DeviceNames[MpFileManagerUIConnect.DeviceList.SelectedIndex];

	// Read if current selected object is folder
	HmiFile.Status.IsFolder := MpFileManagerUIConnect.File.List.Items[HmiFile.Status.SelectedIndex].IsFolder;

	// Control the folder structure when entering and leaving folders
	IF (HmiFile.Commands.EnterFolder) AND MpFileManagerUIConnect.File.List.Items[HmiFile.Status.SelectedIndex].IsFolder THEN
		HmiFile.Commands.EnterFolder := FALSE;
		MpFileManagerUIConnect.File.EnterFolder := TRUE;
		FolderDepthCount := FolderDepthCount + 1;
	ELSE
		HmiFile.Commands.EnterFolder := FALSE;
	END_IF

	IF EDGEPOS(HmiFile.Commands.FolderUp) AND (HmiFile.Status.BackButton > 0) THEN
		HmiFile.Commands.FolderUp := FALSE;
		MpFileManagerUIConnect.File.FolderUp := TRUE;
		FolderDepthCount := FolderDepthCount - 1;
	END_IF

	IF FolderDepthCount > 0 THEN
		HmiFile.Status.BackButton := TRUE;
	ELSE
		HmiFile.Status.BackButton := FALSE;
	END_IF

END_ACTION
```

#### FIFOOperations.st - Implements a first-in-first-out mechanism on one file device
```iecst
ACTION FIFOOperation:

	R_TRIG_CheckStatus(CLK := (MpFileManagerUIConnect.Status = mpFILE_UI_STATUS_CHANGE_DIR) OR
		(MpFileManagerUIConnect.Status = mpFILE_UI_STATUS_CHANGE_DEVICE) OR
		(MpFileManagerUIConnect.Status = mpFILE_UI_STATUS_CREATE));

	IF R_TRIG_CheckStatus.Q OR TON_ScanFolder.Q THEN
		HmiFile.Commands.CheckFolder := TRUE;
	END_IF

	// Autodelete oldest files based on scanning option
    CASE HmiFile.Status.DeleteStep OF

		FILE_DELETE_WAIT:
			// Wait for check the correct device selection
			TON_ScanFolder.IN := (HmiFile.Status.CurrentPage <> 'File_page');
			IF TON_ScanFolder.Q THEN
				TON_ScanFolder.IN := FALSE;
				HmiFile.Status.DeleteStep := FILE_SCAN_FOLDER_WAIT;
			END_IF

		FILE_SCAN_FOLDER_WAIT:
			// Wait for check for old files command
			IF (HmiFile.Commands.CheckFolder = TRUE) AND (MpFileManagerUIConnect.Status = mpFILE_UI_STATUS_IDLE) THEN
				HmiFile.Commands.CheckFolder := FALSE;
				HmiFile.Status.DeleteStep := FILE_SELECT_DEVICE;
				HmiFile.Parameters.OldSortOrder := MpFileManagerUIConnect.File.SortOrder;
			END_IF

		FILE_SELECT_DEVICE:
			//
            IF (HmiFile.Status.DeviceName <> HmiFile.Parameters.Fifo.DeviceName) THEN
				FOR i := 0 TO ((SIZEOF(MpFileManagerUIConnect.DeviceList.DeviceNames)/SIZEOF(MpFileManagerUIConnect.DeviceList.DeviceNames[0])) - 1) DO
        			IF HmiFile.Parameters.Fifo.DeviceName = MpFileManagerUIConnect.DeviceList.DeviceNames[i] THEN
						MpFileManagerUIConnect.DeviceList.SelectedIndex := i;
					END_IF
    			END_FOR
            END_IF

            IF (HmiFile.Status.DeviceName = HmiFile.Parameters.Fifo.DeviceName) AND (MpFileManagerUIConnect.Status = mpFILE_UI_STATUS_IDLE) THEN
                HmiFile.Status.DeleteStep := FILE_SORT_BY_DATE;
            END_IF

		FILE_SORT_BY_DATE:
			// Sort by date so the oldest files are at the end
            IF (MpFileManagerUIConnect.File.SortOrder <> mpFILE_SORT_BY_MOD_TIME_DESC) THEN
                MpFileManagerUIConnect.File.SortOrder := mpFILE_SORT_BY_MOD_TIME_DESC;
            ELSIF (MpFileManagerUIConnect.Status = mpFILE_UI_STATUS_IDLE) THEN
                MpFileManagerUIConnect.File.Refresh := TRUE;
            END_IF

			IF (MpFileManagerUIConnect.Status = mpFILE_UI_STATUS_REFRESH) AND (MpFileManagerUIConnect.File.Refresh = FALSE) THEN
                HmiFile.Status.DeleteStep := FILE_SORT_BY_DATE_WAIT;
            END_IF

       FILE_SORT_BY_DATE_WAIT:
	        // Wait for the file manager to complete sorting change
            IF (MpFileManagerUIConnect.Status = mpFILE_UI_STATUS_IDLE) THEN
                HmiFile.Status.DeleteStep := FILE_CHECK_FOR_FILTER;
            END_IF

		FILE_CHECK_FOR_FILTER:
			// Check which delete filter is active
            IF (HmiFile.Parameters.Fifo.FifoType = FILE_FIFO_NUM_OF_FILES) THEN
                HmiFile.Status.DeleteStep := FILE_SELECT_OLDEST_FILES_0;
            ELSIF (HmiFile.Parameters.Fifo.FifoType = FILE_FIFO_SIZE_OF_FOLDER) THEN
				HmiFile.Status.DeleteStep := FILE_CALC_FOLDER_SIZE;
            END_IF

        FILE_SELECT_OLDEST_FILES_0:
			// Scan and select all file over the filter setting
			IF (MpFileManagerUIConnect.Status = mpFILE_UI_STATUS_IDLE) THEN
				IF MpFileManagerUIConnect.File.PathInfo.FileCount > 1 THEN
           			MpFileManagerUIConnect.File.MultiSelect := TRUE;
				END_IF
				HmiFile.Status.AutoDeleteSelected := 0;
				FOR i := 0 TO ((SIZEOF(HmiFile.Status.FileNames)/SIZEOF(HmiFile.Status.FileNames[0])) - 1) DO
					IF i >= (HmiFile.Parameters.Fifo.MaxNumberOfFiles + MpFileManagerUIConnect.File.PathInfo.FolderCount) THEN
						MpFileManagerUIConnect.File.List.Items[0].IsSelected := FALSE;
						IF (MpFileManagerUIConnect.File.List.Items[i].ItemType <> mpFILE_ITEM_TYPE_NONE) AND NOT MpFileManagerUIConnect.File.List.Items[i].IsFolder THEN
							MpFileManagerUIConnect.File.List.Items[i].IsSelected := TRUE;
							HmiFile.Status.AutoDeleteSelected := HmiFile.Status.AutoDeleteSelected + 1;
						END_IF
					END_IF
				END_FOR

				IF (HmiFile.Status.AutoDeleteSelected > 0) THEN
					HmiFile.Status.DeleteStep := FILE_DELETE_FILES;
				ELSE
					MpFileManagerUIConnect.File.MultiSelect := FALSE;
					HmiFile.Status.DeleteStep := FILE_RESET_SORT_BY;
				END_IF
			END_IF

		FILE_CALC_FOLDER_SIZE:
			// Calculate the overall file size in the open folder
				HmiFile.Status.FolderSize := 0;
				FOR i := 0 TO ((SIZEOF(HmiFile.Status.FileNames)/SIZEOF(HmiFile.Status.FileNames[0])) - 1) DO
					IF MpFileManagerUIConnect.File.List.Items[i].ItemType <> mpFILE_ITEM_TYPE_FOLDER THEN
						HmiFile.Status.FolderSize := HmiFile.Status.FolderSize + UDINT_TO_REAL(MpFileManagerUIConnect.File.List.Items[i].Size);
					END_IF
				END_FOR
				IF (HmiFile.Status.FolderSize > HmiFile.Parameters.Fifo.MaxFolderSize) THEN
					HmiFile.Status.DeleteStep := FILE_SELECT_OLDEST_FILES_1;
				ELSE
					HmiFile.Status.DeleteStep := FILE_RESET_SORT_BY;
				END_IF

		FILE_SELECT_OLDEST_FILES_1:
			// Scan and select all file over the filter setting
			IF (MpFileManagerUIConnect.Status = mpFILE_UI_STATUS_IDLE) THEN
				MpFileManagerUIConnect.File.List.Items[(MpFileManagerUIConnect.File.PathInfo.FileCount - 1)].IsSelected := TRUE;
				HmiFile.Status.DeleteStep := FILE_DELETE_FILES;
			END_IF

		FILE_DELETE_FILES:
			// Set command to delete the selected oldest files
			IF  (MpFileManagerUIConnect.Status = mpFILE_UI_STATUS_IDLE) THEN
				MpFileManagerUIConnect.File.Delete := TRUE;
			END_IF

			IF (MpFileManagerUIConnect.Status = mpFILE_UI_STATUS_DELETE) THEN
				HmiFile.Status.DeleteStep := FILE_CONFIRM_DELETE;
            END_IF

		FILE_CONFIRM_DELETE:
			// Confirm the file delete
            IF (MpFileManagerUIConnect.MessageBox.Type = mpFILE_MSG_CONFIRM_DELETE) THEN
                MpFileManagerUIConnect.MessageBox.Confirm := TRUE;
            ELSIF (MpFileManagerUIConnect.Status = mpFILE_UI_STATUS_IDLE) AND (MpFileManagerUIConnect.MessageBox.LayerStatus = 1) THEN
				IF (HmiFile.Parameters.Fifo.FifoType = FILE_FIFO_SIZE_OF_FOLDER) THEN
                	HmiFile.Status.DeleteStep := FILE_CALC_FOLDER_SIZE;
				ELSE
					HmiFile.Status.DeleteStep := FILE_RESET_SORT_BY;
					MpFileManagerUIConnect.File.MultiSelect := FALSE;
				END_IF
            END_IF

		FILE_RESET_SORT_BY:
			// Restore old sort order
            IF (MpFileManagerUIConnect.File.SortOrder <> HmiFile.Parameters.OldSortOrder) THEN
                MpFileManagerUIConnect.File.SortOrder := HmiFile.Parameters.OldSortOrder;
            ELSIF (MpFileManagerUIConnect.Status = mpFILE_UI_STATUS_IDLE) THEN
                MpFileManagerUIConnect.File.Refresh := TRUE;
				HmiFile.Status.DeleteStep := FILE_RESET_SORT_BY_WAIT;
            END_IF

		FILE_RESET_SORT_BY_WAIT:
			// Wait for file manager to complete restoring previous sorting mode
            IF (MpFileManagerUIConnect.Status = mpFILE_UI_STATUS_REFRESH) OR (MpFileManagerUIConnect.Status = mpFILE_UI_STATUS_IDLE) THEN
                HmiFile.Status.DeleteStep := FILE_DELETE_WAIT;
				IF (MpFileManagerUIConnect.MessageBox.Type = mpFILE_MSG_BUSY) THEN
					MpFileManagerUIConnect.MessageBox.Confirm := TRUE;
				END_IF
            END_IF
	END_CASE

	// Timer to scan file device in intervals
	TON_ScanFolder(PT := DINT_TO_TIME(HmiFile.Parameters.Fifo.ScanInterval * 60000));

END_ACTION
```

### Program Logical/Infrastructure/Recipe/RecipeMgr

#### RecipeMgr.typ
```iecst
(*Structure types*)

TYPE
	RecipeHmiInterfaceType : 	STRUCT  (*Structure to hold commands, parameters and status from the HMI*)
		Commands : RecipeCommandsType; (*Structure to hold the commands from the HMI*)
		Parameters : RecipeParametersType; (*Structure to hold the parameters for the HMI*)
		Status : RecipeStatusType; (*Structure to hold status information from the mapp View HMI*)
	END_STRUCT;
	RecipeCommandsType : 	STRUCT  (*Structure to hold the commands from the HMI*)
		LoadRecipe : BOOL; (*Load recipe*)
		SaveSelectedRecipe : BOOL; (*Save the selected recipe (which is not necessarily the active recipe)*)
		CreateRecipe : BOOL; (*Create recipe*)
		ImportFromUSB : BOOL; (*Import from USB device*)
		ExportToUSB : BOOL; (*Export to USB device*)
	END_STRUCT;
	RecipeParametersType : 	STRUCT  (*Structure to hold the parameters for the HMI*)
		Category : STRING[30]; (*Current category*)
		DeviceDataProvider : ARRAY[0..MAX_IDX_FILE_DEV]OF STRING[100]; (*File device data provider*)
		DeviceName : STRING[50]; (*Selected file device name*)
		FileName : STRING[255]; (*Recipe file name*)
		TableConfig : STRING[120]; (*Table configuration *)
	END_STRUCT;
	RecipeStatusType : 	STRUCT  (*Structure to hold status information from the mapp View HMI*)
		HMIcommand : RecipeHmiStepEnum; (*State machine step for HMI commands*)
		LastLoadedConfigRecipe : STRING[255]; (*Last loaded configuration recipe*)
		LastLoadedProductRecipe : STRING[255]; (*Last loaded product recipe*)
		ActiveRecipe : STRING[255]; (*The name of the active recipe*)
		LastMaxSelection : UINT; (*The previous maximum number of recipes*)
		LastSelectedIndex : UINT; (*The previous selected index*)
		LastStatus : MpRecipeUIStatusEnum; (*The previous UI status*)
		CopyStep : RecipeCopyStepEnum; (*State machine step for copying a recipe to/from a USB drive*)
		CategoryDropdown : STRING[50]; (*Category dropdown value*)
		EditDialogOpened : BOOL; (*Flag that the edit dialog box was opened*)
		CreateDialogOpened : BOOL; (*Flag that the create dialog box was opened*)
		PreviousRecipe : STRING[80]; (*Name of the previous recipe*)
		FileDuplicate : BOOL; (*Recipe file already exists, warn the user.*)
		FilesAvailable : BOOL; (*Control access to widget when no files are available*)
	END_STRUCT;
	ParametersType : 	STRUCT  (*Demo / starter structure for machine parameters*)
		AddParametersHere1 : BOOL; (*Add your parameteres here *)
		AddParametersHere2 : STRING[80]; (*Add your parameteres here *)
		AddParametersHere3 : REAL; (*Add your parameteres here *)
		AddParametersHere4 : REAL; (*Add your parameteres here *)
		AddParametersHere5 : REAL; (*Add your parameteres here *)
	END_STRUCT;
	MachineSettingsType : 	STRUCT  (*Demo / starter structure for machine configuration settings*)
		AddMachineSettingsHere1 : USINT; (*Add your settings here*)
		AddMachineSettingsHere2 : DINT; (*Add your settings here*)
		AddMachineSettingsHere3 : BOOL; (*Add your settings here*)
		AddMachineSettingsHere4 : REAL; (*Add your settings here*)
		AddMachineSettingsHere5 : UINT; (*Add your settings here*)
	END_STRUCT;
END_TYPE

(*Enumerations*)

TYPE
	RecipeCopyStepEnum :
		( (*State machine step for copying a recipe to/from a USB drive*)
		REC_COPY_WAIT := 0, (*Wait state*)
		REC_COPY_TO_USB, (*Copy to USB*)
		REC_COPY_FROM_USB, (*Copy from USB*)
		REC_COPY_BUSY (*Busy*)
		);
	RecipeHmiStepEnum :
		( (*State machine step for HMI commands*)
		REC_HMI_WAIT, (*Wait*)
		REC_HMI_LOAD, (*Load recipe*)
		REC_HMI_SAVE, (*Save recipe*)
		REC_HMI_CREATE (*Create recipe*)
		);
END_TYPE
```

#### RecipeMgr.var
```iecst
(*Function Blocks*)
VAR
	MpRecipe_0 : MpRecipeXml; (*MpRecipe instance*)
	MpRecipeRegPar_PreviewPar : MpRecipeRegPar; (*MpRecipeRegPar instance for ParametersPreview variable*)
	MpRecipeRegPar_PreviewCfg : MpRecipeRegPar; (*MpRecipeRegPar instance for MachineSettingsPreview*)
	MpRecipeUI_0 : MpRecipeUI; (*MpRecupeUI instance*)
	MpFileManagerUI_0 : MpFileManagerUI; (*MpFileManagerUI instance*)
	DTGetTime_0 : DTGetTime; (*DTGetTime instance*)
	DirCreate_0 : DirCreate; (*DirCreate instance*)
END_VAR
(*Constants*)
VAR CONSTANT
	MAX_IDX_FILE_DEV : USINT := MAX_IDX_USB_DEV_LIST + 1; (*Maximum number of  file devices *)
	DEFAULT_PARAMETERS : STRING[12] := 'Default.par'; (*Default parameters recipe file name*)
	DEFAULT_MACHINE_CONFIGURATION : STRING[12] := 'Machine.mcfg'; (*Default machine configuration recipe file name*)
END_VAR
VAR
	PARAMETERS_RECIPE : STRING[50] := 'Parameters'; (*Value of the DropDownBox selection for the Parameters category*)
	MACHINE_CONFIGURATION_RECIPE : STRING[50] := 'Machine Configuration'; (*Value of the DropDownBox selection for the Machine Configuration category*)
END_VAR
VAR CONSTANT
	LOCAL_FOLDER : STRING[10] := 'Recipe'; (*Folder name on the file device for Recipe files*)
END_VAR
(*Structure Types*)
VAR
	HmiRecipe : RecipeHmiInterfaceType; (*HMI interface structure*)
	Parameters : ParametersType; (*Machine parameters. Used by the machine at runtime*)
	ParametersEdit : {REDUND_UNREPLICABLE} ParametersType; (*Machine parameters edit structure. Enables you to edit a recipe that is not currently active*)
	ParametersPreview : ParametersType; (*Machine parameters preview structure. Registered to the recipe. Enables you to preview a recipe that is not currently active.*)
	MachineSettings : MachineSettingsType; (*Machine settings. Used by the machine at runtime.*)
	MachineSettingsEdit : MachineSettingsType; (*Machine settings edit structure. Enables you to edit a recipe that is not currently active*)
	MachineSettingsPreview : MachineSettingsType; (*Machine settings preview structure. Registered to the recipe. Enables you to preview a recipe that is not currently active. *)
	MpRecipeUIConnect : MpRecipeUIConnectType; (*MpRecipeUI connection to the HMI*) (*ParameterFileStep : INT;*)
	MpRecipeUISetup : MpRecipeUISetupType; (*MpRecipeUI setup connection to the HMI*) (*ParameterFileStep : INT;*)
	MpFileManagerUIConnect : MpFileManagerUIConnectType; (*File manager connection to the HMI*)
	Header : MpRecipeXmlHeaderType; (*Header information*)
END_VAR
(*Variables*)
VAR
	i : USINT; (*Index to loop through file devices*)
	temp : STRING[260]; (*Temporary recipe name, used to check for duplicates when creating a new recipe*)
END_VAR
```

#### RecipeMgr.st
```iecst
//***********************************************************************
// Copyright: B&R Industrial Automation GmbH
// Author: B&R Industrial Automation GmbH
// Created: Jan 1, 2022
// Description: Tasks for recipe control.
//***********************************************************************

PROGRAM _INIT

	// Create folder for this component on the user file device
	DirCreate_0(enable := TRUE, pDevice := ADR('UserPartition'), pName := ADR(LOCAL_FOLDER));

	// Check if folder already exist and if so disabled the function block call
	IF DirCreate_0.status = fiERR_DIR_ALREADY_EXIST THEN
		DirCreate_0(enable := FALSE);
	END_IF

	// Initialize mapp function blocks
	// By default, the Framework sets up an XML recipe system. To swtich to the CSV format, refer to the "Change Recipe Format"
	// page in the AS Help (GUID 2052b3a5-f59b-45f9-9fcd-3289c93401af)
	MpRecipeUISetup.Confirmation.RecipeDelete := TRUE;
	MpRecipeUISetup.RecipeListSize := 10;
	MpRecipeUISetup.RecipeListScrollWindow := 0;
	MpRecipeUISetup.AutoLoadHeader := TRUE;
	MpRecipeUIConnect.New.FileName := 'newRecipe';
	MpRecipeUIConnect.Recipe.Filter := '*par';
	MpRecipeUI_0.MpLink := ADR(gMpLinkRecipeXml);
	MpRecipeUI_0.Enable := TRUE;
	MpRecipeUI_0.UIConnect := ADR(MpRecipeUIConnect);
	MpRecipeUI_0.UISetup := MpRecipeUISetup;
	MpRecipeUI_0();

	HmiRecipe.Parameters.Category := PARAMETERS_CATEGORY;
	HmiRecipe.Parameters.DeviceDataProvider[0] := '{"value":"mappRecipeFiles","text":"CF/PLC"}';
	HmiRecipe.Parameters.DeviceName := 'mappRecipeFiles';
	MpRecipe_0.MpLink := ADR(gMpLinkRecipeXml);
	MpRecipe_0.Enable := TRUE;
	MpRecipe_0.Category := ADR(HmiRecipe.Parameters.Category);
	MpRecipe_0.DeviceName := ADR(HmiRecipe.Parameters.DeviceName);
    MpRecipe_0.FileName := ADR(HmiRecipe.Parameters.FileName);
	MpRecipe_0.Header := ADR(Header);

	// Wait for MpRecipe_0 to activate. This must be active before you can call the RegPar function blocks, which is below.
	WHILE NOT(MpRecipe_0.Active OR MpRecipe_0.Error) DO
		MpRecipe_0();
	END_WHILE

	// Register the preview variables to the recipe. These preview variables are a buffer between the recipe system and the
	// variables used at runtime on the machine (Parameters, MachineSettings). By using these preview variables, you can
	// preview and edit a recipe on the HMI without actually loading it to the machine. For more details, refer to the
	// "Recipe System Design" page in the AS Help (GUID 3ccd7409-0b52-4bbc-a93a-4010f6db414c).

    MpRecipeRegPar_PreviewPar.MpLink := ADR(gMpLinkRecipeXml);
	MpRecipeRegPar_PreviewPar.Enable := TRUE;
	MpRecipeRegPar_PreviewPar.PVName := ADR('RecipeMgr:ParametersPreview');
	MpRecipeRegPar_PreviewPar.Category := ADR(PARAMETERS_CATEGORY);
	MpRecipeRegPar_PreviewPar();

	MpRecipeRegPar_PreviewCfg.MpLink := ADR(gMpLinkRecipeXml);
	MpRecipeRegPar_PreviewCfg.Enable := TRUE;
	MpRecipeRegPar_PreviewCfg.PVName := ADR('RecipeMgr:MachineSettingsPreview');
	MpRecipeRegPar_PreviewCfg.Category := ADR(MACHINE_CONFIGURATION_CATEGORY);
	MpRecipeRegPar_PreviewCfg();

	// Wait for RegPar function blocks to activate. These must be active before you can load a recipe,
	// which is further down in the Initialization program.
	WHILE NOT(MpRecipeRegPar_PreviewPar.Active OR MpRecipeRegPar_PreviewPar.Error) DO
		MpRecipeRegPar_PreviewPar();
	END_WHILE
	WHILE NOT(MpRecipeRegPar_PreviewCfg.Active OR MpRecipeRegPar_PreviewCfg.Error) DO
		MpRecipeRegPar_PreviewCfg();
	END_WHILE

	// Load default Machine Settings recipe
	HmiRecipe.Parameters.Category := MACHINE_CONFIGURATION_CATEGORY;
	HmiRecipe.Parameters.FileName := DEFAULT_MACHINE_CONFIGURATION;
	MpRecipe_0.Load := TRUE;
	WHILE NOT(MpRecipe_0.CommandDone OR MpRecipe_0.Error) DO
		MpRecipe_0();
    END_WHILE
	MachineSettings := MachineSettingsPreview;

	MpRecipe_0.ErrorReset := MpRecipe_0.Error;
	MpRecipe_0.Load := FALSE;
	MpRecipe_0();

	// Load default Parameter recipe
	HmiRecipe.Parameters.Category := PARAMETERS_CATEGORY;
	HmiRecipe.Parameters.FileName := DEFAULT_PARAMETERS;
	HmiRecipe.Status.PreviousRecipe := DEFAULT_PARAMETERS;
	MpRecipe_0.Load := TRUE;
	WHILE NOT(MpRecipe_0.CommandDone OR MpRecipe_0.Error) DO
		MpRecipe_0();
	END_WHILE
	Parameters := ParametersPreview;

	HmiRecipe.Status.LastLoadedProductRecipe := DEFAULT_PARAMETERS;
	HmiRecipe.Status.LastLoadedConfigRecipe := DEFAULT_MACHINE_CONFIGURATION;
	MpRecipe_0.ErrorReset := MpRecipe_0.Error;
	MpRecipe_0.Load := FALSE;
	MpRecipe_0();

    // Trigger update notification so that the initial parameters are copied to the process
    // might not be necessary.*****
	MpRecipe_0.UpdateNotification := TRUE;

	// Init Filemanager for exporting/importing files
	MpFileManagerUI_0.Enable := TRUE;
	MpFileManagerUI_0.MpLink := ADR(gMpLinkFileManagerUIRecipe);
	MpFileManagerUI_0.UIConnect := ADR(MpFileManagerUIConnect);
	MpFileManagerUI_0.UISetup.FileListSize := SIZEOF(MpFileManagerUIConnect.File.List.Items) / SIZEOF(MpFileManagerUIConnect.File.List.Items[0]);
	MpFileManagerUIConnect.DeviceList.DeviceNames[0] := 'mappRecipeFiles';
	MpFileManagerUIConnect.DeviceList.DeviceNames[1] := '';
	MpFileManagerUI_0();

	HmiRecipe.Status.HMIcommand := REC_HMI_WAIT;

END_PROGRAM

PROGRAM _CYCLIC

	// Call actions
	FormatDeviceDataProvider;
	LoadPreview;
	RecipeHMIcommands;
	FileCopyOperation;

	// Reset commands on MpRecipe FUB
	IF MpRecipe_0.CommandDone THEN
		MpRecipe_0.Load := FALSE;
		MpRecipe_0.Save := FALSE;
		// Set update notification for machine category
	//	IF ((brsstrcmp(ADR(HmiRecipe.Parameters.Category), ADR(MACHINE_CONFIGURATION_CATEGORY)) = 0) AND (MpRecipe_0.Save = TRUE)) THEN
		IF ((brsstrcmp(ADR(HmiRecipe.Status.CategoryDropdown), ADR(MACHINE_CONFIGURATION_CATEGORY)) = 0) AND (MpRecipe_0.Save = TRUE)) THEN
			MpRecipe_0.UpdateNotification := TRUE;
		ELSE
			MpRecipe_0.UpdateNotification := FALSE;
			HmiRecipe.Parameters.Category := PARAMETERS_CATEGORY;
			HmiRecipe.Parameters.FileName := 'Default.par';
		END_IF
		END_IF

	// Error reset
	IF NOT MpRecipe_0.Error THEN
		MpRecipe_0.ErrorReset := FALSE;
	END_IF

	IF NOT MpRecipeUI_0.Error THEN
		MpRecipeUI_0.ErrorReset := FALSE;
	END_IF

	// Assign MpLinks
	MpRecipe_0.MpLink := ADR(gMpLinkRecipeXml);
	MpRecipeUI_0.MpLink := ADR(gMpLinkRecipeXml);
	MpFileManagerUI_0.MpLink := ADR(gMpLinkFileManagerUIRecipe);
	MpRecipeRegPar_PreviewPar.MpLink := ADR(gMpLinkRecipeXml);
	MpRecipeRegPar_PreviewCfg.MpLink := ADR(gMpLinkRecipeXml);

	// Call function blocks
	MpRecipe_0();
	MpRecipeUI_0();
	MpFileManagerUI_0();
	MpRecipeRegPar_PreviewPar();
	MpRecipeRegPar_PreviewCfg();

END_PROGRAM

PROGRAM _EXIT

	// Disable the function blocls to unlink the MpLinks
	MpRecipe_0.Enable := FALSE;
	MpRecipeUI_0.Enable := FALSE;
	MpRecipeRegPar_PreviewPar.Enable := FALSE;
	MpRecipeRegPar_PreviewCfg.Enable := FALSE;
	MpFileManagerUI_0.Enable := FALSE;

	// Call function blocks
	MpRecipe_0();
	MpRecipeUI_0();
	MpRecipeRegPar_PreviewPar();
	MpRecipeRegPar_PreviewCfg();
	MpFileManagerUI_0();

END_PROGRAM
```

### Program Logical/Infrastructure/SysServices/IoBrowser (IEC)

#### Variables.var - Local variables
```iecst
(*Io process related variables*)
VAR
	GatIoForcingHandler_0 : GatIoForcingHandler; (*Function block for Io handling (browser & forcing)*)
	IoModules : ARRAY[0..gatMAX_IDX_IO_MODULES] OF GatIoModulesType;
	IoChannelTemp : REFERENCE TO GatIoChannelType;
	IoChannel : REFERENCE TO GatIoChannelType;
END_VAR
(*Helper variables for mappView*)
VAR
	StationList : ARRAY[0..gatMAX_IDX_IO_MODULES] OF STRING[80];
	ModuleList : ARRAY[0..gatMAX_IDX_IO_MODULES] OF STRING[80];
	IoChannelList : ARRAY[0..gatMAX_IDX_IO_CHANNELS] OF STRING[80];
	IoPvList : ARRAY[0..gatMAX_IDX_IO_CHANNELS] OF STRING[80];
	IoValueListString : ARRAY[0..gatMAX_IDX_IO_CHANNELS] OF STRING[20];
	IoValueList : ARRAY[0..gatMAX_IDX_IO_CHANNELS] OF DINT;
	StationIdx : UINT;
	ModuleIdx : UINT;
	ChannelIdx : UINT;
	SelectedStation : STRING[80];
	SelectedStationIndex : UINT;
	LastSelectedStationIndex : UINT;
	SelectedModule : UINT;
	LastSelectedModule : UINT;
	SelectedChannel : UINT;
	LastSelectedChannel : UINT;
	TableConfigChannels : STRING[200];
	TableConfigStations : STRING[200];
	TableConfig : STRING[200];
	TempStationPath : STRING[80];
	LastModuleInvisible : BOOL;
END_VAR
```

### Program Logical/Infrastructure/SysServices/ProcessConfig

#### Variables.var
```iecst
VAR
	MC_BR_ProcessConfig_AX : MC_BR_ProcessConfig; (*Function block to read and write the axis configuration*)
	MC_BR_ProcessConfig_ACP : MC_BR_ProcessConfig; (*Function block to read and write the ACOPOS configuration*)
	BaseAxConfig : ARRAY[0..1] OF McCfgAxType; (*Acopos configuration*)
	AcpAxConfig : ARRAY[0..1] OF McCfgAcpAxType; (*Acopos configuration*)
	SelectedAxis : USINT; (*Selected Axis index*)
	AxFeatures1 : ARRAY[0..2] OF STRING[255]; (*Axis features*)
	AxFeatures2 : ARRAY[0..2] OF STRING[255]; (*Axis features*)
	State : UINT; (*Read/Write state machine status*)
	ReadConfig : BOOL; (*Read config command*)
	WriteConfig : BOOL; (*Write Acopos config command*)
	SuccessRead : BOOL; (*Read config succeeded*)
	ErrorRead : BOOL; (*Read config failed*)
	ErrorWrite : BOOL; (*Write config failed*)
	SuccessWrite : BOOL; (*Write config succeeded*)
	SysReboot : BOOL;
	MpRecipeRegPar_M : ARRAY[0..3] OF MpRecipeRegPar;
	MC_BR_ProcessParam_ACP : MC_BR_ProcessParam;
END_VAR
```

#### Main.st
```iecst
//*********************************************************************************
//* Copyright: B&R Industrial Automation GmbH
//* This task let's the OEM change the ACOPOS configuration via the HMI
//*********************************************************************************

PROGRAM _INIT
	// FUB configuration: MC_BR_ProcessConfig for persistent configuration changes, MC_BR_ProcessParam for online configuration changes
    MC_BR_ProcessConfig_ACP.DataType := mcCFG_ACP_AX;

	AcpAxConfig[0].AxisFeatures.FeatureReference.DataAddress := ADR(AxFeatures1);
	AcpAxConfig[0].AxisFeatures.FeatureReference.NumberOfArrayElements := 3;
	AcpAxConfig[1].AxisFeatures.FeatureReference.DataAddress := ADR(AxFeatures2);
	AcpAxConfig[1].AxisFeatures.FeatureReference.NumberOfArrayElements := 3;

	MC_BR_ProcessConfig_AX.DataType := mcCFG_AX;

	MC_BR_ProcessParam_ACP.ExecutionMode := mcEM_IMMEDIATELY;
	MC_BR_ProcessParam_ACP.Mode := mcPPM_WRITE;

	// Register "Machine" category PVs
	MpRecipeRegPar_M[0].MpLink := ADR(gMpLinkRecipeXml);
	MpRecipeRegPar_M[0].Enable := TRUE;
	MpRecipeRegPar_M[0].Category := ADR('Machine Configuration');
	MpRecipeRegPar_M[0].PVName := ADR('ProcessCon:AcpAxConfig');
	MpRecipeRegPar_M[1].MpLink := ADR(gMpLinkRecipeXml);
	MpRecipeRegPar_M[1].Enable := TRUE;
	MpRecipeRegPar_M[1].Category := ADR('Machine Configuration');
	MpRecipeRegPar_M[1].PVName := ADR('ProcessCon:BaseAxConfig');
	MpRecipeRegPar_M[2].MpLink := ADR(gMpLinkRecipeXml);
	MpRecipeRegPar_M[2].Enable := TRUE;
	MpRecipeRegPar_M[2].Category := ADR('Machine Configuration');
	MpRecipeRegPar_M[2].PVName := ADR('ProcessCon:sAxFeatures1');
	MpRecipeRegPar_M[3].MpLink := ADR(gMpLinkRecipeXml);
	MpRecipeRegPar_M[3].Enable := TRUE;
	MpRecipeRegPar_M[3].Category := ADR('Machine Configuration');
	MpRecipeRegPar_M[3].PVName := ADR('ProcessCon:sAxFeatures2');

	// Activate RegPar FUBs
	WHILE NOT MpRecipeRegPar_M[0].Active DO
		MpRecipeRegPar_M[0]();
	END_WHILE
	WHILE NOT MpRecipeRegPar_M[1].Active DO
		MpRecipeRegPar_M[1]();
	END_WHILE
	WHILE NOT MpRecipeRegPar_M[2].Active DO
		MpRecipeRegPar_M[2]();
	END_WHILE
	WHILE NOT MpRecipeRegPar_M[3].Active DO
		MpRecipeRegPar_M[3]();
	END_WHILE

	// Trigger first read
	ReadConfig := TRUE;
	State := 0;
END_PROGRAM

PROGRAM _CYCLIC
	// Read/Write state machine
	CASE State OF
        0:
            // Idle
			IF MpRecipeRegPar_M[0].UpdateNotification THEN
				// Reset the address of sAxFeatures1/2
				AcpAxConfig[0].AxisFeatures.FeatureReference.DataAddress := ADR(AxFeatures1);
				AcpAxConfig[0].AxisFeatures.FeatureReference.NumberOfArrayElements := 3;
				AcpAxConfig[1].AxisFeatures.FeatureReference.DataAddress := ADR(AxFeatures2);
				AcpAxConfig[1].AxisFeatures.FeatureReference.NumberOfArrayElements := 3;

				// Write the configuration
				SelectedAxis := 0;
				WriteConfig := TRUE;
				ReadConfig := FALSE;
			ELSIF ReadConfig THEN
				// Set axis dependend configuration name
				IF SelectedAxis = 0 THEN
					brsstrcpy(ADR(MC_BR_ProcessConfig_ACP.Name), ADR('IF1.ST1/DriveConfiguration/Channel1'));
				ELSE
					brsstrcpy(ADR(MC_BR_ProcessConfig_ACP.Name), ADR('IF1.ST1/DriveConfiguration/Channel2'));
				END_IF
				AcpAxConfig[0].AxisFeatures.FeatureReference.DataAddress := ADR(AxFeatures1);
				AcpAxConfig[0].AxisFeatures.FeatureReference.NumberOfArrayElements := 3;
				AcpAxConfig[1].AxisFeatures.FeatureReference.DataAddress := ADR(AxFeatures2);
				AcpAxConfig[1].AxisFeatures.FeatureReference.NumberOfArrayElements := 3;

				MC_BR_ProcessConfig_ACP.DataAddress := ADR(AcpAxConfig[SelectedAxis]);
				MC_BR_ProcessConfig_AX.DataAddress := ADR(BaseAxConfig[SelectedAxis]);
				// Start loading
				MC_BR_ProcessConfig_ACP.Mode := mcPCM_LOAD;
				MC_BR_ProcessConfig_ACP.Execute := TRUE;
				ErrorRead := FALSE;
				SuccessRead := FALSE;
				State := 10;
			ELSIF WriteConfig THEN
				// Set axis dependend configuration name
				IF SelectedAxis = 0 THEN
					brsstrcpy(ADR(MC_BR_ProcessConfig_ACP.Name), ADR('IF1.ST1/DriveConfiguration/Channel1'));
					MC_BR_ProcessParam_ACP.Component := ADR(gAxisMaster);
				ELSE
					brsstrcpy(ADR(MC_BR_ProcessConfig_ACP.Name), ADR('IF1.ST1/DriveConfiguration/Channel2'));
					MC_BR_ProcessParam_ACP.Component := ADR(gAxisSlave);
				END_IF
				MC_BR_ProcessConfig_ACP.DataAddress := ADR(AcpAxConfig[SelectedAxis]);
				MC_BR_ProcessConfig_AX.DataAddress := ADR(BaseAxConfig[SelectedAxis]);
                MC_BR_ProcessParam_ACP.DataAddress := ADR(AcpAxConfig[SelectedAxis].MechanicalElements);
                // mcCFG_ACP_AX is not supported yet, therefore, transfer mech elements and homing parameters in two steps
				MC_BR_ProcessParam_ACP.DataType := mcCFG_ACP_MECH_ELM;
				// Copy direct homing position into the used homing mode, HMI is bound to direct homing position
				CASE AcpAxConfig[SelectedAxis].Homing.Mode.Type OF
					mcAHM_ABS:
						AcpAxConfig[SelectedAxis].Homing.Mode.Absolute.Position := AcpAxConfig[SelectedAxis].Homing.Mode.Direct.Position;
					mcAHM_ABS_CORR:
						AcpAxConfig[SelectedAxis].Homing.Mode.AbsoluteCorrection.Position := AcpAxConfig[SelectedAxis].Homing.Mode.Direct.Position;
					mcAHM_ABS_SW:
						AcpAxConfig[SelectedAxis].Homing.Mode.AbsoluteSwitch.Position := AcpAxConfig[SelectedAxis].Homing.Mode.Direct.Position;
					mcAHM_BLK_LAG_ERR:
						AcpAxConfig[SelectedAxis].Homing.Mode.BlockLagError.Position := AcpAxConfig[SelectedAxis].Homing.Mode.Direct.Position;
                    mcAHM_BLK_TORQ:
                        AcpAxConfig[SelectedAxis].Homing.Mode.BlockTorque.Position := AcpAxConfig[SelectedAxis].Homing.Mode.Direct.Position;
					mcAHM_DIST_C_MARKS:
						AcpAxConfig[SelectedAxis].Homing.Mode.DistanceCodedMarks.Position := AcpAxConfig[SelectedAxis].Homing.Mode.Direct.Position;
					mcAHM_DIST_C_MARKS_CORR:
						AcpAxConfig[SelectedAxis].Homing.Mode.DistanceCodedMarksCorrection.Position := AcpAxConfig[SelectedAxis].Homing.Mode.Direct.Position;
					mcAHM_LIM_SW:
						AcpAxConfig[SelectedAxis].Homing.Mode.LimitSwitch.Position := AcpAxConfig[SelectedAxis].Homing.Mode.Direct.Position;
					mcAHM_SW_GATE:
						AcpAxConfig[SelectedAxis].Homing.Mode.SwitchGate.Position := AcpAxConfig[SelectedAxis].Homing.Mode.Direct.Position;
				END_CASE;
				MC_BR_ProcessConfig_ACP.Mode := mcPCM_SAVE;
				MC_BR_ProcessConfig_ACP.Execute := TRUE;
				MC_BR_ProcessConfig_AX.Mode := mcPCM_SAVE;
				MC_BR_ProcessConfig_AX.Execute := TRUE;
				MC_BR_ProcessParam_ACP.Execute := TRUE;
				ErrorWrite := FALSE;
				SuccessWrite := FALSE;
				State := 20;
			END_IF

        10:
            // Read config
			IF MC_BR_ProcessConfig_ACP.Done OR MC_BR_ProcessConfig_ACP.Error THEN
				MC_BR_ProcessConfig_ACP.Execute := FALSE;
				// Copy homing position into the direct homing position, HMI is bound to direct homing position
				CASE AcpAxConfig[SelectedAxis].Homing.Mode.Type OF
					mcAHM_ABS:
						AcpAxConfig[SelectedAxis].Homing.Mode.Direct.Position := AcpAxConfig[SelectedAxis].Homing.Mode.Absolute.Position;
					mcAHM_ABS_CORR:
						AcpAxConfig[SelectedAxis].Homing.Mode.Direct.Position := AcpAxConfig[SelectedAxis].Homing.Mode.AbsoluteCorrection.Position;
					mcAHM_ABS_SW:
						AcpAxConfig[SelectedAxis].Homing.Mode.Direct.Position := AcpAxConfig[SelectedAxis].Homing.Mode.AbsoluteSwitch.Position;
					mcAHM_BLK_LAG_ERR:
						AcpAxConfig[SelectedAxis].Homing.Mode.Direct.Position := AcpAxConfig[SelectedAxis].Homing.Mode.BlockLagError.Position;
					mcAHM_BLK_TORQ:
						AcpAxConfig[SelectedAxis].Homing.Mode.Direct.Position := AcpAxConfig[SelectedAxis].Homing.Mode.BlockTorque.Position;
					mcAHM_DIST_C_MARKS:
						AcpAxConfig[SelectedAxis].Homing.Mode.Direct.Position := AcpAxConfig[SelectedAxis].Homing.Mode.DistanceCodedMarks.Position;
					mcAHM_DIST_C_MARKS_CORR:
						AcpAxConfig[SelectedAxis].Homing.Mode.Direct.Position := AcpAxConfig[SelectedAxis].Homing.Mode.DistanceCodedMarksCorrection.Position;
					mcAHM_LIM_SW:
						AcpAxConfig[SelectedAxis].Homing.Mode.Direct.Position := AcpAxConfig[SelectedAxis].Homing.Mode.LimitSwitch.Position;
					mcAHM_SW_GATE:
						AcpAxConfig[SelectedAxis].Homing.Mode.Direct.Position := AcpAxConfig[SelectedAxis].Homing.Mode.SwitchGate.Position;
				END_CASE;
				brsstrcpy(ADR(MC_BR_ProcessConfig_AX.Name), ADR(AcpAxConfig[SelectedAxis].AxisReference.Name));
				MC_BR_ProcessConfig_AX.Mode := mcPCM_LOAD;
				MC_BR_ProcessConfig_AX.Execute := TRUE;
				ErrorRead := FALSE;
				SuccessRead := TRUE;
				State := 11;
			ELSIF MC_BR_ProcessConfig_ACP.Error THEN
				MC_BR_ProcessConfig_ACP.Execute := FALSE;
				ErrorRead := TRUE;
				SuccessRead := FALSE;
				ReadConfig := FALSE;
				State := 0;
			END_IF

        11:
            // Read axis config
			IF MC_BR_ProcessConfig_AX.Done OR MC_BR_ProcessConfig_AX.Error THEN
				MC_BR_ProcessConfig_AX.Execute := FALSE;
				ErrorRead := MC_BR_ProcessConfig_AX.Error;
				SuccessRead := NOT bErrorRead;
				IF SelectedAxis = 0 THEN
					SelectedAxis := 1;
				ELSE
					ReadConfig := FALSE;
				END_IF
				State := 0;
			END_IF

        20:
            // Write config
			IF (MC_BR_ProcessConfig_ACP.Done OR MC_BR_ProcessConfig_ACP.Error)
				AND (MC_BR_ProcessConfig_AX.Done OR MC_BR_ProcessConfig_AX.Error)
				AND (MC_BR_ProcessParam_ACP.Done OR MC_BR_ProcessParam_ACP.Error) THEN
				MC_BR_ProcessConfig_ACP.Execute := FALSE;
				MC_BR_ProcessConfig_AX.Execute := FALSE;
				MC_BR_ProcessParam_ACP.Execute := FALSE;
				ErrorWrite := MC_BR_ProcessConfig_ACP.Error OR MC_BR_ProcessConfig_AX.Error OR MC_BR_ProcessParam_ACP.Error;
				SuccessWrite := NOT ErrorWrite;
				State := 21;
			END_IF

        21:
            // Write Homing config
			MC_BR_ProcessParam_ACP.DataAddress := ADR(AcpAxConfig[SelectedAxis].Homing);// mcCFG_ACP_AX is not supported yet, therefore, transfer mech elements and homing parameters in two steps
			MC_BR_ProcessParam_ACP.DataType := mcCFG_ACP_HOME;
			MC_BR_ProcessParam_ACP.Execute := TRUE;
			IF MC_BR_ProcessParam_ACP.Done OR MC_BR_ProcessParam_ACP.Error THEN
				MC_BR_ProcessParam_ACP.Execute := FALSE;
				ErrorWrite := bErrorWrite OR MC_BR_ProcessParam_ACP.Error;
				SuccessWrite := NOT bErrorWrite;
				State := 0;
				// Update the second axis, or finish
				IF SelectedAxis = 0 THEN
					SelectedAxis := 1;
				ELSE
					WriteConfig := FALSE;
				END_IF
			END_IF
	END_CASE;

	// PLC reboot
	IF SysReboot THEN
		SYSreset(TRUE, 1);
	END_IF

	// Function block calls
	MC_BR_ProcessConfig_ACP();
	MC_BR_ProcessConfig_AX();
	MC_BR_ProcessParam_ACP();
	MpRecipeRegPar_M[0]();
	MpRecipeRegPar_M[1]();
	MpRecipeRegPar_M[2]();
	MpRecipeRegPar_M[3]();
END_PROGRAM

PROGRAM _EXIT
	// Release mplink
	MpRecipeRegPar_M[0].Enable := FALSE;
	MpRecipeRegPar_M[1].Enable := FALSE;
	MpRecipeRegPar_M[2].Enable := FALSE;
	MpRecipeRegPar_M[3].Enable := FALSE;
	MpRecipeRegPar_M[0]();
	MpRecipeRegPar_M[1]();
	MpRecipeRegPar_M[2]();
	MpRecipeRegPar_M[3]();
END_PROGRAM
```

### Program Logical/Infrastructure/SysServices/SysServs

#### Types.typ
```iecst
TYPE
	CpuIoMapType : 	STRUCT
		SerialNumber_CPU : UDINT;
		ModuleID_CPU : UINT;
		HardwareVariant : UINT;
		FirmwareVersion : UINT;
		TemperatureCPU : INT;
		TemperatureENV : INT;
		SystemTime : DINT;
		TerminalOK : BOOL;
		TerminalStatus : USINT;
		TerminalTemperatureCPU : INT;
		TerminalLoadCPU0 : USINT;
		TerminalLoadCPU1 : USINT;
	END_STRUCT;
	LanguageSelect : 	STRUCT
		LanguageSelection : ARRAY[0..1]OF STRING[80] := ['en','de'];
		SelectedIndex : INT := 0;
	END_STRUCT;
	EthConfigType : 	STRUCT
		Ip : STRING[15];
		Gateway : STRING[15];
		SubnetMask : STRING[15];
		Device : STRING[20];
	END_STRUCT;
	ClientInfoType : 	STRUCT
		userId : STRING[40];
		ipAddress : STRING[15];
		activityCount : USINT;
		languageId : STRING[10];
		isValid : BOOL;
		currentPageId : STRING[40];
		measurementSystemId : STRING[10];
	END_STRUCT;
END_TYPE
```

#### Variables.var
```iecst
(********************************************************************
 * COPYRIGHT -- Bernecker + Rainer
 ********************************************************************
 * Program: FolderHandling
 * File: FolderHandling.var
 * Author: Bernecker + Rainer
 * Created: December , 2020
 ********************************************************************
 * Local variables of program Visualization Control
 ********************************************************************)
(*Variable Declaration*)
VAR
	EthConfig : EthConfigType; (*Ethernet configuration*)
	CpuIoMap : CpuIoMapType; (*Cpu IO Mapping*)
	CfgGetSubnetMask_0 : CfgGetSubnetMask; (*GetSubnetMask*)
	CfgGetIPAddr_0 : CfgGetIPAddr; (*GetIPAddr*)
	CfgGetDefaultGateway_0 : CfgGetDefaultGateway; (*GetDefaultGateway*)
	CfgSetSubnetMask_0 : CfgSetSubnetMask; (*GetSubnetMask*)
	CfgSetIPAddr_0 : CfgSetIPAddr; (*GetIPAddr*)
	CfgSetDefaultGateway_0 : CfgSetDefaultGateway; (*GetDefaultGateway*)
	CurrentMode : STRING[80]; (*Current Mode(Simulation/Runtime)*)
	Simulation : BOOL; (*Simulation Mode Flag(1: Simulation 0: Runtime)*)
	ReadEthConfig : BOOL;
	WriteEthConfig : BOOL;
	DTStructureSetTime_0 : DTStructureGetTime;
	DTStructureGetTime_0 : DTStructureSetTime;
	DateTimeCfg : DTStructure; (*Date Structure*)
	ClientInfo : ARRAY[0..MAX_IDX_CLIENTS] OF ClientInfoType;
END_VAR
VAR CONSTANT
	MAX_IDX_CLIENTS : USINT := 3;
END_VAR
```

#### Main.st
```iecst
//*********************************************************************************
//* Copyright: B&R Industrial Automation GmbH
//* Created:   30. Sep 2020/08:00
//* Description: Tasks FOR Visualization control. The HMI handling is done in this task.
//********************************************************************************

PROGRAM _INIT
	// Insert code here

    brsstrcpy(ADR(EthConfig.Device), ADR('IF2'));

    // Configure Ethernet configuration function blocks
    CfgGetIPAddr_0.pDevice := ADR(EthConfig.Device);
    CfgGetDefaultGateway_0.pDevice := ADR(EthConfig.Device);
    CfgGetSubnetMask_0.pDevice := ADR(EthConfig.Device);
    CfgGetIPAddr_0.pIPAddr := ADR(EthConfig.Ip);
    CfgGetDefaultGateway_0.pGateway := ADR(EthConfig.Gateway);
    CfgGetSubnetMask_0.pSubnetMask := ADR(EthConfig.SubnetMask);
    CfgGetIPAddr_0.Len := 16;
    CfgGetDefaultGateway_0.Len := 16;
    CfgGetSubnetMask_0.Len := 16;
    CfgSetIPAddr_0.pDevice := ADR(EthConfig.Device);
	CfgSetDefaultGateway_0.pDevice := ADR(EthConfig.Device);
	CfgSetSubnetMask_0.pDevice := ADR(EthConfig.Device);
	CfgSetIPAddr_0.pIPAddr := ADR(EthConfig.Ip);
	CfgSetDefaultGateway_0.pGateway := ADR(EthConfig.Gateway);
	CfgSetSubnetMask_0.pSubnetMask := ADR(EthConfig.SubnetMask);
	CfgSetIPAddr_0.Option := 1;
	CfgSetDefaultGateway_0.Option := 1;
	CfgSetSubnetMask_0.Option := 1;

	// Read ETHERNET information after booting
	ReadEthConfig := TRUE;

	// Configure Get/Set time function blocks
	DTStructureGetTime_0.pDTStructure := ADR(DateTimeCfg);
	DTStructureSetTime_0.pDTStructure := ADR(DateTimeCfg);

	// Client info
	ClientInfo[0].activityCount := 0;
END_PROGRAM

PROGRAM _CYCLIC
	// Read ethernet information from target
	IF ReadEthConfig THEN
		CfgGetIPAddr_0.enable := TRUE;
		CfgGetDefaultGateway_0.enable := TRUE;
		CfgGetSubnetMask_0.enable := TRUE;
		ReadEthConfig := FALSE;
	END_IF
	// Write ethernet information to target
	IF WriteEthConfig THEN
		CfgSetIPAddr_0.enable := TRUE;
		CfgSetDefaultGateway_0.enable := TRUE;
		CfgSetSubnetMask_0.enable := TRUE;
		WriteEthConfig := FALSE;
	END_IF

	// Call ethernet configuration related function blocks
	CfgGetIPAddr_0();
	CfgGetDefaultGateway_0();
	CfgGetSubnetMask_0();
	CfgSetIPAddr_0();
	CfgSetDefaultGateway_0();
	CfgSetSubnetMask_0();

	// Reset the enable inputs when done
	IF (CfgGetIPAddr_0.status <> ERR_FUB_BUSY) AND (CfgGetIPAddr_0.status <> ERR_FUB_ENABLE_FALSE) THEN
		CfgGetIPAddr_0.enable := FALSE;
	END_IF
	IF (CfgGetDefaultGateway_0.status <> ERR_FUB_BUSY) AND (CfgGetDefaultGateway_0.status <> ERR_FUB_ENABLE_FALSE) THEN
		CfgGetDefaultGateway_0.enable := FALSE;
	END_IF
	IF (CfgGetSubnetMask_0.status <> ERR_FUB_BUSY) AND (CfgGetSubnetMask_0.status <> ERR_FUB_ENABLE_FALSE) THEN
		CfgGetSubnetMask_0.enable := FALSE;
	END_IF
	IF (CfgSetIPAddr_0.status <> ERR_FUB_BUSY) AND (CfgSetIPAddr_0.status <> ERR_FUB_ENABLE_FALSE) THEN
		CfgSetIPAddr_0.enable := FALSE;
	END_IF
	IF (CfgSetDefaultGateway_0.status <> ERR_FUB_BUSY) AND (CfgSetDefaultGateway_0.status <> ERR_FUB_ENABLE_FALSE) THEN
		CfgSetDefaultGateway_0.enable := FALSE;
	END_IF
	IF (CfgSetSubnetMask_0.status <> ERR_FUB_BUSY) AND (CfgSetSubnetMask_0.status <> ERR_FUB_ENABLE_FALSE) THEN
		CfgSetSubnetMask_0.enable := FALSE;
	END_IF

	// Reset time function block enable commands
	IF (DTStructureGetTime_0.status <> ERR_FUB_BUSY) AND (DTStructureGetTime_0.status <> ERR_FUB_ENABLE_FALSE) THEN
		DTStructureGetTime_0.enable := FALSE;
	END_IF
	IF (DTStructureSetTime_0.status <> ERR_FUB_BUSY) AND (DTStructureSetTime_0.status <> ERR_FUB_ENABLE_FALSE) THEN
		DTStructureSetTime_0.enable := FALSE;
	END_IF

	// Call time configuration function blocks
	DTStructureGetTime_0();
	DTStructureSetTime_0();

	IF CpuIoMap.SerialNumber_CPU = 0 THEN
		CurrentMode := 'Simulation Mode' ;
		Simulation := TRUE ;
	ELSE
		CurrentMode := 'Runtime Mode' ;
		Simulation := FALSE ;
	END_IF

END_PROGRAM

PROGRAM _EXIT
	// Insert code here

END_PROGRAM
```

### Library Logical/Infrastructure/TS_UnitTest/Libraries/UnitTest (ANSIC, version 2.01.0) - Static library for UnitTest programs written in ANSI C /C++

#### UnitTest.h
```c
/*****************************************************************************
 * COPYRIGHT (C) BERNECKER + RAINER
 *****************************************************************************
 * Library:  UnitTest
 * File:     UnitTest.h
 * Author:   B+R
 *****************************************************************************
 * Description: Static library for UnitTest programs written in ANSI C /C++
 *
 * Add the path "\Logical\TS_UnitTest\Libraries\UnitTest\" to the
 * "Additional include directories" in the tab "Build" (PLC Properties)
 ******************************************************************************/

#ifndef	__UNITTEST_H__
#define	__UNITTEST_H__
#ifdef __cplusplus
extern "C"
{
#endif
#include <bur/plctypes.h>

#ifndef NULL
#define	NULL	0
#endif
#include "include/Test.h"

#include "include/TestCase.h"
#include "include/TestListener.h"
#include "include/TestResult.h"
#include "include/TestCaller.h"

#include "include/AssertImpl.h"
#include "include/HelperMacro.h"
#include "include/utRunner.h"

/* function is a test case */
#define _TEST 			static testStatusEnum

/* function is a setup */
#define _SETUP_TEST 	static testStatusEnum 	setupTest

/* function is a teardown */
#define _TEARDOWN_TEST 	static testStatusEnum 	teardownTest

/* function is a setup for whole test set */
#define _SETUP_SET		static testStatusEnum	setupSet

/* function is a teardown for whole test set */
#define _TEARDOWN_SET 	static testStatusEnum	teardownSet

/* function is a cyclic handler for test set */
#define _CYCLIC_SET		static void 			cyclicSetCaller

/* Skipped test case */
#define SKIP_TEST  		_TEST
/* Skip all test cases of set */
#define SKIP_TEST_SET

/* Dummies for smart edit autocompletion.
See AssertImpl.h for real macros used by the compiler  */
#ifdef _SMART_EDIT_DUMMY_

/* String comparison.
Returns true if the strings are equal. */
BOOL TEST_ASSERT_EQUAL_STRING(char *expected,char  *actual);
/* Wstring comparison.
Returns true if the WSTRINGS are equal. */
BOOL TEST_ASSERT_EQUAL_WSTRING(unsigned short *expected,unsigned short *actual);
 /* Compares two memory blocks.
Returns true if [size] bytes are equal. */
BOOL TEST_ASSERT_EQUAL_MEM(void *expected, void *actual,UDINT size);
/* Compares integer values. Usable for all integer types.
Avoid comparison of unsigned with signed types.
Returns true if they are equal.
Note: If different, values are reported as DINT values in the test report */
BOOL TEST_ASSERT_EQUAL_INT(expected, actual);

/* Compares REAL values with delta = (expected * TEST_FLOAT_PRECISION).
Returns true if (difference <= delta) */
BOOL TEST_ASSERT_EQUAL_REAL(REAL expected,REAL actual);
/* Compares REAL values with explicit delta.
Returns true if (difference <= delta) */
BOOL TEST_ASSERT_REAL_WITHIN(REAL delta, REAL expected, REAL actual);
/* Compares LREAL values with delta = (expected * TEST_DOUBLE_PRECISION).
Returns true if (difference <= delta) */
BOOL TEST_ASSERT_EQUAL_LREAL(LREAL expected,LREAL  actual);
/* Compares LREAL values with explicit delta.
Returns true if (difference <= delta) */
BOOL TEST_ASSERT_LREAL_WITHIN(LREAL delta, LREAL expected, LREAL actual);

/* Compares float values with delta = (expected * TEST_FLOAT_PRECISION).
Returns true if (difference <= delta) */
BOOL TEST_ASSERT_EQUAL_FLOAT(float expected, float actual);
/* Compares float values with explicit delta.
Returns true if (difference <= delta) */
BOOL TEST_ASSERT_FLOAT_WITHIN(float delta, float expected, float actual);
/* Compares double values with delta = (expected * TEST_DOUBLE_PRECISION).
Returns true if (difference <= delta) */
BOOL TEST_ASSERT_EQUAL_DOUBLE(double expected, double actual);
/* Compares double values with explicit delta.
Returns true if (difference <= delta) */
BOOL TEST_ASSERT_DOUBLE_WITHIN(double delta, double expected, double actual);

/* Returns true if pointer is null */
BOOL TEST_ASSERT_NULL(void *pointer);
/* Returns true if pointer is not null */
BOOL TEST_ASSERT_NOT_NULL(void *pointer);
/* Returns true, if condition evals to  true */
BOOL TEST_ASSERT_MESSAGE(condition, char *message);
/* Returns true, if condition evals to  true */
BOOL TEST_ASSERT(condition);

/* Returns always false */
BOOL TEST_FAIL(char *message);

/* Add a note to the test report */
void TEST_INFO(char *message);
/* Add a note with location information to the test report */
void TEST_INFO_POS(char *message);

#ifdef __cplusplus
/* Test if expression throws given exception.
Catches all other exceptions as failure.
Note: Available for C++ only */
void TEST_ASSERT_THROW(expression, type);

/* Fails if expression throws any exceptions.
Note: Available for C++ only*/
void TEST_ASSERT_NO_THROW(expression);
#endif

/* Adds a test function with description to the Testfixture.
See UNITTEST_FIXTURES() */
void new_TestFixture(char *name, _TEST function);

/* Adds a test function with description to the Testfixture.
This test will be skipped
See UNITTEST_FIXTURES() */
void skipTestFixture(char *name, _TEST function);

/* Defines the order of test cases.
Should look like this
UNITTEST_FIXTURES(fixtures)
{
	new_TestFixture("test_1",test_1),
	new_TestFixture("test_2",test_2),
	new_TestFixture("test_3",test_3)
}
*/
void UNITTEST_FIXTURES(fixtures)

/* Standard UnitTest caller without any setup / teardown methods*/
void UNITTEST_CALLER_TEST(caller, char *name, fixtures);

/* Standard UnitTest caller with macro setup / teardown for tests*/
void UNITTEST_CALLER_BASIC(caller, char *name, fixtures);

/* UnitTest caller with macro setup / teardown for tests and test set */
void UNITTEST_CALLER_SET(caller, char *name, fixtures);

/* UnitTest caller with macro setup / teardown for tests and test set and cylic*/
void UNITTEST_CALLER_COMPLETE(caller, char *name, fixtures);

/* UnitTest caller with explicit setup / teardown for suite */
void UNITTEST_CALLER_SET_EXPLICIT(caller,name,setupTest,teardownTest,fixtures, setupSuite, teardownSuite);

/* UnitTest caller with explicit setup / teardown for suite and cylic */
void UNITTEST_CALLER_COMPLETE_EXPLICIT(caller,name,setupTest,teardownTest,fixtures, setupSuite, teardownSuite, cyclicCaller);

/* Adds a test set with description to the fixture of test sets.
See UNITTEST_TESTSET_FIXTURES() */
void new_TestSet(testcaller);

/* Defines the order of test sets.
Should look like this
UNITTEST_TESTSET_FIXTURES(fixtures)
{
	new_TestSet(testSet_1),
	new_TestSet(testSet_2),
	new_TestSet(testSet_3)
}*/
void UNITTEST_TESTSET_FIXTURES(fixtures);

/* Defines the test set list handling structure*/
void UNTITTEST_TESTSET_HANDLER();

#endif /*_SMART_EDIT_DUMMY_*/

/*
 Use to declare Test set for use in list of test sets of test programm
 See usage in autogeneratedFile.c / FixtureOfTestSets.c
*/
#define UNITTEST_TESTSET_DECLARATION 	extern const TestCaller

/* Default factor for precision used to test if REAL / float values  are equal.
(0.00001f) */
#define TEST_FLOAT_PRECISION 	(0.00001f)
/* Default factor for precision used to test if LREAL / double values  are equal.
(1e - 12f) */
#define TEST_DOUBLE_PRECISION 	(1e-12f)

#if (__GNUC__ != 6) || (__GNUC_MINOR__ != 3) || (__GNUC_PATCHLEVEL__ != 0)
#error UnitTest is compiled with GCC version 6.3.0. To use UnitTest switch GCC version to 6.3.0 or import a different solution package
#endif

#define UNIT_TEST_LIBRARY_VERSION  			"2.01.0"

#ifdef __cplusplus
};
#endif

#include "include/asserts.hpp"

#endif/*__UNITTEST_H__*/
```

- THIRDPARTYLICENSEREADME (not shown)

#### AssertImpl.h - Available asserts
```c
/*
* Author: 		B+R
* Contents of this file are modified and extended
*/

/*
 * COPYRIGHT AND PERMISSION NOTICE
 *
 * Copyright (c) 2003 Embedded Unit Project
 *
 * All rights reserved.
 *
 * Permission is hereby granted, free of charge, to any person obtaining
 * a copy of this software and associated documentation files (the
 * "Software"), to deal in the Software without restriction, including
 * without limitation the rights to use, copy, modify, merge, publish,
 * distribute, and/or sell copies of the Software, and to permit persons
 * to whom the Software is furnished to do so, provided that the above
 * copyright notice(s) and this permission notice appear in all copies
 * of the Software and that both the above copyright notice(s) and this
 * permission notice appear in supporting documentation.
 *
 * THE SOFTWARE IS PROVIDED "AS IS", WITHOUT WARRANTY OF ANY KIND,
 * EXPRESS OR IMPLIED, INCLUDING BUT NOT LIMITED TO THE WARRANTIES OF
 * MERCHANTABILITY, FITNESS FOR A PARTICULAR PURPOSE AND NONINFRINGEMENT
 * OF THIRD PARTY RIGHTS. IN NO EVENT SHALL THE COPYRIGHT HOLDER OR
 * HOLDERS INCLUDED IN THIS NOTICE BE LIABLE FOR ANY CLAIM, OR ANY
 * SPECIAL INDIRECT OR CONSEQUENTIAL DAMAGES, OR ANY DAMAGES WHATSOEVER
 * RESULTING FROM LOSS OF USE, DATA OR PROFITS, WHETHER IN AN ACTION OF
 * CONTRACT, NEGLIGENCE OR OTHER TORTIOUS ACTION, ARISING OUT OF OR IN
 * CONNECTION WITH THE USE OR PERFORMANCE OF THIS SOFTWARE.
 *
 * Except as contained in this notice, the name of a copyright holder
 * shall not be used in advertising or otherwise to promote the sale,
 * use or other dealings in this Software without prior written
 * authorization of the copyright holder.
 *
 * $Id: AssertImpl.h,v 1.6 2003/09/16 11:09:53 arms22 Exp $
 */

#ifndef	__ASSERTIMPL_H__
#define	__ASSERTIMPL_H__

#ifdef	__cplusplus
extern "C" {
#endif

#include <bur/plctypes.h>

/* Increments failure counter and outputs failure text*/
void addFailure(const char *msg, unsigned long line, const char *file);
/* Increments passed counter*/
void addPassed(const char *msg, unsigned long line, const char *file);
/* Outputs informational text*/
void addInfo(const char *msg, unsigned long line, const char *file);
/* Increments abort counter, aborts current test set, outputs abort text.
    Existing teardown methods will be called before leaving the test set */
void addAbort(const char *msg, unsigned long line, const char *file);

BOOL assertImplementationInt(int expected,int actual, unsigned long line, const char *file);
BOOL assertImplementationCStr(const char *expected,const char *actual, unsigned long line, const char *file);
BOOL assertImplementationDoublesWithin(const double delta,	const double expected,	const double actual,	unsigned long line, const char *file);
BOOL assertImplementationFloatsWithin(const float delta,	const float expected,	const float actual,	unsigned long line, const char *file);
BOOL assertImplementationWStr(const unsigned short *expected,const unsigned short *actual, unsigned long line, const char *file);
BOOL assertCondition(BOOL condition, const char *message,  unsigned long line, const char *file);
BOOL assertImplementationMem(void *expected ,void  *actual, unsigned long  size, unsigned long line, const char *file);

#define TEST_ASSERT_EQUAL_STRING(expected,actual)\
	assertImplementationCStr(expected,actual,__LINE__,__FILE__)

#define TEST_ASSERT_EQUAL_WSTRING(expected,actual)\
	assertImplementationWStr(expected,actual,__LINE__,__FILE__)

#define TEST_ASSERT_EQUAL_MEM(expected,actual,size)\
	assertImplementationMem(expected,actual,size,__LINE__,__FILE__)

#define TEST_ASSERT_EQUAL_INT(expected,actual)\
	assertImplementationInt(expected, actual,__LINE__,__FILE__)

#define TEST_ASSERT_NULL(pointer)\
	TEST_ASSERT_MESSAGE(pointer == NULL,#pointer " was not null.")

#define TEST_ASSERT_NOT_NULL(pointer)\
	TEST_ASSERT_MESSAGE(pointer != NULL,#pointer " was null.")

#define TEST_ASSERT_MESSAGE(condition, message)\
	assertCondition(condition,message,__LINE__,__FILE__)

#define TEST_ASSERT(condition) \
	assertCondition(condition, #condition,__LINE__,__FILE__)

#define TEST_FAIL(message)\
	assertCondition(0, message,__LINE__,__FILE__)

#define TEST_ASSERT_EQUAL_FLOAT(expected, actual)   		\
	assertImplementationFloatsWithin(\
									 (float)(expected) * (float)TEST_FLOAT_PRECISION, \
									 (float)(expected), (float)(actual), \
									 (unsigned long) __LINE__, __FILE__)

#define TEST_ASSERT_FLOAT_WITHIN(delta, expected, actual)	 \
	assertImplementationFloatsWithin(\
									 (float)(delta), \
									 (float)(expected), (float)(actual), \
									 (unsigned long) __LINE__, __FILE__)

#define TEST_ASSERT_EQUAL_DOUBLE(expected, actual)           \
	assertImplementationDoublesWithin(\
									  (double)(expected) * (double)TEST_DOUBLE_PRECISION,\
									  (double)(expected), (double)(actual), \
									  (unsigned long) __LINE__, __FILE__)

#define TEST_ASSERT_DOUBLE_WITHIN(delta, expected, actual)    \
	assertImplementationDoublesWithin(\
									  (double)(delta),\
									  (double)(expected), (double)(actual), \
									  (unsigned long) __LINE__, __FILE__)

	/* IEC data types*/
#define TEST_ASSERT_EQUAL_REAL(expected, actual)     		TEST_ASSERT_EQUAL_FLOAT(expected, actual)
#define TEST_ASSERT_REAL_WITHIN(delta, expected, actual)    TEST_ASSERT_FLOAT_WITHIN(delta, expected, actual)

#define TEST_ASSERT_EQUAL_LREAL(expected, actual)  			TEST_ASSERT_EQUAL_DOUBLE(expected, actual)
#define TEST_ASSERT_LREAL_WITHIN(delta, expected, actual)	TEST_ASSERT_DOUBLE_WITHIN(delta, expected, actual)

#define TEST_INFO(message)		addInfo(message,0,0);
#define TEST_INFO_POS(message)	addInfo(message,__LINE__,__FILE__)

	/* Returns and signals completion.
	Note: This is a return statement*/
#define TEST_DONE 				return ut_DONE

	/* Returns and signals that this call is not yet completed. Will be called again in next cycle.
	Note: This is a conditional return statement*/
#define TEST_BUSY 				return ut_BUSY

	/* If condition is true: Returns and signals that this call is not yet completed. Will be called again in next cycle.
	Note: This is a conditional return statement */
#define TEST_BUSY_CONDITION(condition) 				if(condition) { 	TEST_BUSY; }
	/* If condition is true: Returns and signals that this call is not yet completed. Will be called again in next cycle.
	A message is reported.
	Note: This is a conditional return statement*/
#define TEST_BUSY_CONDITION_MSG(condition, msg) 	if(condition) {	TEST_INFO( msg );  TEST_BUSY; }

	/* Returns and signals abortion of current test set.
	No further test case of this set will be executed.
	If available teardown methods will be called before test set is left.
	Note: This is a return statement*/
#define TEST_ABORT								{addAbort("Test set aborted.",__LINE__,__FILE__);} return ut_ABORT

	/* Returns and signals that this test case is aborted.
	No further test case of this set will be executed.
	If available teardown methods will be called before test set is left.
	A message is reported.
	Note: This is a return statement*/
#define TEST_ABORT_MSG(message)					{addAbort(message,__LINE__,__FILE__);} return ut_ABORT

	/* If condition is true: Returns and signals that this test case is aborted.
	No further test case of this set will be executed.
	If available teardown methods will be called before test set is left.
	Note: This is a conditional return statement*/
#define TEST_ABORT_CONDITION(condition) 				if(condition) { 	TEST_ABORT; }

	/* If condition is true: Returns and signals that this test case is aborted.
	No further test case of this set will be executed.
	If available teardown methods will be called before test set is left.
	A message is reported
	Note: This is a conditional return statement*/
#define TEST_ABORT_CONDITION_MSG(condition, msg) 		if(condition) { TEST_ABORT_MSG(msg); }

#ifdef	__cplusplus
}
#endif

#endif/*__ASSERTIMPL_H__*/
```
